(* CODESYS project Almost_done.export

Project tree, tasks and I/O mapping:
  Device : CODESYS Control Win V3 x64, 3S - Smart Software Solutions GmbH, version 3.5.17.0
    application Application
      libraries: Standard, * (System); VisuDialogs, * (System)
      task MainTask (cyclic, interval t#20ms, priority 1) calls PLC_PRG
      task VISU_TASK (cyclic, interval 100 ms, priority 31) calls VisuElems.Visu_Prg
      global variables GVL
      global variables HMI
      global variables OPC
      function block Assembly [ST]
      function block Crane [ST]
      function block ExitMagazine [ST]
      function FillWarehouseArray [ST]
      function FindFreePlace [ST]
      function block PalletizerElevator [ST]
      program PLC_PRG [ST]
      function Round [ST]
      function SetArrayToZero [ST]
      function block ThreeAxis [ST]
      function block TwoAxisLogic [ST]
      function WhereIsMaterial [ST]
      Symbols
      visualisation Assembly
      visualisation Menu
      visualisation Package_Reload
      visualisation Palletizer
      visualisation QA
      visualisation Warehosue_1
      visualisation Warehouse_2
*)

// Device/Application/GVL
VAR_GLOBAL
	Warehouse1Array : ARRAY[1..54] OF BOOL;
	Warehouse1ArrayMaterial  : ARRAY[1..54] OF INT;
	Warehouse2Array : ARRAY[1..54] OF INT ;
	Warehouse2ArrayMaterial  : ARRAY[1..54] OF INT;
	PalletizerArray : ARRAY[0..12] OF BOOL;
END_VAR

// Device/Application/HMI
{attribute 'qualified_only'}
VAR_GLOBAL
	GoingQA : BOOL;
	Emitter1Color : INT := 16;
	Emitter2Color : INT := 16;
	WantedMaterial1 : INT;
	Pick1 : BOOL;
	WantedMaterial2 : INT;
	Pick2 : BOOL;
	ScreenColor : INT := 0;
	EmittMaterials : BOOL := TRUE;
	
	oElevator1Forward : BOOL;
	oPalletizer1Open  : BOOL;
	oPalletizer1Push  : BOOL;
	oPalletizer1Clamp  : BOOL;
	oPalletizer1Forward  : BOOL;
	oPalletizer1ElevatorUp  : BOOL;
	oPalletizer1ChainForward  : BOOL;
	oPalletizer1ElevatorDown : BOOL;
	oPalletizer1ElevatorMoveToMax  : BOOL;
	oPalletizerConv  : BOOL;
	oPalletizerSupplyConv  : BOOL;
	oPalletizerSupplyLightConv  : BOOL;
	oPalletsTowardElevator  : BOOL;
	oPalletizer1Turn  : BOOL;
END_VAR

// Device/Application/OPC
{attribute 'qualified_only'}
VAR_GLOBAL
	// This part includes 2 first machines center and surroundings machines
	iAtAssembledConvEntry : BOOL;
	iAtAssemledPosition : BOOL;
	iMachine1Exit : BOOL;
	iMachine2Exit : BOOL;
	iMachine1Entry : BOOL;
	iMachine2Entry : BOOL;
	iMachiningCenter1Error : BOOL;
	iMachiningCenter2Error : BOOL;
	iMachiningCenter1IsBusy : BOOL;
	iMachiningCenter1Opened : BOOL;
	iMachiningCenter2IsBusy : BOOL;
	iMachiningCenter2Opened : BOOL;
	iMachiningCenter1Progress : DINT;
	iMachiningCenter2Progress : DINT;
	iRightPositioner2Clamped : BOOL;
	iRightPositioner1Clamped : BOOL;
	iRightPositioner1OnPlace : BOOL;
	iRightPositioner2OnPlace : BOOL;
	iRightPositioner3Clamped : BOOL;
	iRightPositioner3OnPlace : BOOL;
	iTwoAxis1Grabbed : BOOL;
	iTwoAxis1MovingX : BOOL;
	iTwoAxis1MovingZ : BOOL;
	iVisionSenserPart1 : DINT;
	iVisionSenserPart2 : DINT;
	
	oAssembledMaterialConv : BOOL;
	oBaseMaterialConv1 : BOOL;
	oBaseMaterialConv2 : BOOL;
	oEmitter1Base : INT;
	oEmitter1Emit : BOOL;
	oEmitter1Part : INT;
	oEmitter2Base : INT;
	oEmitter2Emit : BOOL;
	oEmitter2Part : INT;
	oLiquidMaterialConv1 : BOOL;
	oLiquidMaterialConv2 : BOOL;
	oMachiningCenter1Product : BOOL;
	oMachiningCenter2Product : BOOL;
	oRawMaterialSupply1 : BOOL;
	oRawMaterialSupply2 : BOOL;
	oRightPositioner2Clamp : BOOL;
	oRightPositioner1Clamp : BOOL;
	oRightPositioner1Raise : BOOL;
	oRightPositioner2Raise : BOOL;
	oRightPositioner3Clamp : BOOL;
	oRightPositioner3Raise : BOOL;
	oTwoAxis1X : BOOL;
	oTwoAxis1Z : BOOL;
	oTwoAxis1Grab : BOOL;
	
	//This part include second and third twoAxis pick and place, QA and surroundings conveyors, and first warehouse conveyros
	iAtAssemblyLoadEntry : BOOL;
	iAtCrane1Entry : BOOL;
	iAtCurveConv1Exit : BOOL;
	iAtCurveConv1Entry : BOOL;
	iAtFirstwarehouseCurveConv2Exit : BOOL;
	iAtFirstwarehouseCurveConv2Entry : BOOL;
	iAtPusher : BOOL;
	iAtQACurveEntry : BOOL;
	iAtQAEntry : BOOL;
	iAtQAExit : BOOL;
	iAtWeightConvExit : BOOL;
	iAtWeightConvEntry : BOOL;
	iAtTurntable1Entry : BOOL;
	iAtTurntable1ExitQA : BOOL;
	iAtTurntable1ExitNormal : BOOL;
	iPusher1Back : BOOL;
	iPusher2Back : BOOL;
	iPusher3Back : BOOL;
	iPusher1Front : BOOL;
	iPusher2Front : BOOL;
	iPusher3Front : BOOL;
	iTurntable1Back : BOOL;
	iTurntable1Front : BOOL;
	iTurntable1AtZero : BOOL;
	iTurntable1AtNinety : BOOL;
	iTwoAxis2Grabbed : BOOL;
	iTwoAxis2MovingX : BOOL;
	iTwoAxis3Grabbed : BOOL;
	iTwoAxis3MovingX : BOOL;
	iTwoAxis3MovingZ : BOOL;
	iTwoAxis2MovingZ : BOOL;
	iVisionSensor1 : BOOL;
	iVisionSensor2 : BOOL;
	iWeightConv : REAL;
	iAtQALightConvExit : BOOL;
	iAtElevator2Entry : BOOL;
	iElevator2LeftLimit : BOOL;
	iElevator2RightLimit : BOOL;
	iElevator2CurrentPoint : REAL;
	
	oFirstWarehouseConv1 : BOOL;
	oFirstWarehouseConv3 : BOOL;
	oFirstWarehouseConvLoad : BOOL;
	oFirstWarehouseCurveConv2 : BOOL;
	oPalletAndBoxConv1 : BOOL;
	oPalletAndBoxConv3 : BOOL;
	oPalletAndBoxCurveConv2 : BOOL;
	oPusher1 : BOOL;
	oPusher2 : BOOL;
	oPusher3 : BOOL;
	oQAConv2 : BOOL;
	oQACurveConv : BOOL;
	oQALightConv1 : BOOL;
	oQALightConv2 : BOOL;
	oQALightConv3 : BOOL;
	oQALightConv4 : BOOL;
	oTurntable1Turn : BOOL;
	oTurntable1Forward : BOOL;
	oTurntable1Backward : BOOL;
	oTwoAxis2X : BOOL;
	oTwoAxis2Z : BOOL;
	oTwoAxis3X : BOOL;
	oTwoAxis3Z : BOOL;
	oTwoAxis2Grab : BOOL;
	oTwoAxis3Grab : BOOL;
	oWeightConvBackward : BOOL;
	oWeightConvToward : BOOL;
	oElevator2Forward : BOOL;
	oElevator2SetPoint : REAL;
	oQAConv1 : BOOL;
	
	//This part includes two cranes and conveyor betweeen them
	iAtCrane1Exit : BOOL;
	iAtCrane2Exit : BOOL;
	iAtExitWarehouseExit : BOOL;
	iAtTurntable2Exit : BOOL;
	iAtTurntable2Entry : BOOL;
	iAtTurntable2ExitWarehouse1 : BOOL;
	iAtTurntable2ExitWarehouse2 : BOOL;
	iCrane1AtStart : BOOL;
	iCrane2AtStart : BOOL;
	iCrane1MovingX : BOOL;
	iCrane1MovingZ : BOOL;
	iCrane2MovingX : BOOL;
	iCrane2MovingZ : BOOL;
	iCrane1MidLimit : BOOL;
	iCrane2MidLimit : BOOL;
	iCrane1LeftLimit : BOOL;
	iCrane2LeftLimit : BOOL;
	iCrane1RightLimit : BOOL;
	iCrane2RightLimit : BOOL;
	iTurntable2Back : BOOL;
	iTurntable2Front : BOOL;
	iTurntable2Atzero : BOOL;
	iTurntable2AtNinety : BOOL;
	
	oCrane1Left : BOOL;
	oCrane1Lift : BOOL;
	oCrane2Left : BOOL;
	oCrane2Lift : BOOL;
	oCrane1Right : BOOL;
	oCrane2Right : BOOL;
	oCrane1TargetPosition : INT;
	oCrane2TargetPosition : INT;
	oExitWarehouseConv1 : BOOL;
	oExitWarehouseConv2 : BOOL;
	oFirstWarehouseConvLoadOpposite : BOOL;
	oSecondWarehouseLoadConvOpposite : BOOL;
	oTowardFirstWarehouse : BOOL;
	oTowardSecondWarehouse : BOOL;
	oTurntable2Turn : BOOL;
	oTurntable2Forward : BOOL;
	oTurntable2Backward : BOOL;

	//this part include Box Pick and Place, and conveyors till elevator
	iAtBoxSupplyCurveConv2Exit : BOOL;
	iAtBoxSupplyCurveConv2Entry : BOOL;
	iAtBoxSupplyEnter : BOOL;
	iAtElevatorEntry : BOOL;
	iAtLoadEmptyBoxEntry : BOOL;
	iAtLoadEmptyBoxExit : BOOL;
	iAtPalletDestinationEntry : BOOL;
	iAtPalletDestinationExit : BOOL;
	iAtSecondWarehouseCurveConv3Exit : BOOL;
	iAtSecondWarehouseCurveConv3Entry : BOOL;
	iAtSecondWarehouseConv5 : BOOL;
	iBigBox : BOOL;
	iMidBox : BOOL;
	iPickPlace1Rotated : BOOL;
	iPickPlace1CurrentX : REAL;
	iPickPlace1CurrentY : REAL;
	iPickPlace1CurrentZ : REAL;
	iPickPlace1BoxDetected : BOOL;
	iSmallBox : BOOL;
	
	oBoxSupplyConv1 : BOOL;
	oBoxSupplyConv3 : BOOL;
	oBoxSupplyCurveConv2 : BOOL;
	oEmptyBoxConvSupply : BOOL;
	oPickPlace1X : REAL;
	oPickPlace1Y : REAL;
	oPickPlace1Z : REAL;
	oPickPlace1Grab : BOOL;
	oSecondWarehouseConv1 : BOOL;
	oSecondWarehouseConv12 : BOOL;
	oSecondWarehouseConv2 : BOOL;
	oSecondWarehouseConv4 : BOOL;
	oSecondWarehouseConv5 : BOOL;
	oSecondWarehouseCurveConv3 : BOOL;
	
	//Palletizer
	iAtElevatorUpEntry : BOOL;
	iAtPalletizerChainEntry : BOOL;
	iAtPalletizerConvEntry : BOOL;
	iAtPalletizerEntry : BOOL;
	iPalletizer1Clamped : BOOL;
	iPalletizer1Opening : BOOL;
	iPalletizer1Pushing : BOOL;
	iPalletizer1ElevatorBack : BOOL;
	iPalletizer1ElevatorFront : BOOL;
	iPalletizer1ElevatorMoving : BOOL;
	
	oPalletizer1Open : BOOL;
	oPalletizer1Push : BOOL;
	oPalletizer1Turn : BOOL;
	oPalletizer1Clamp : BOOL;
	oPalletizer1Forward : BOOL;
	oPalletizer1ElevatorUp : BOOL;
	oPalletizer1ChainForward : BOOL;
	oPalletizer1ElevatorDown : BOOL;
	oPalletizer1ChainBackward : BOOL;
	oPalletizer1ElevatorMoveToMax : BOOL;
	oPalletizerConv : BOOL;
	oPalletizerSupplyConv : BOOL;
	oPalletizerSupplyLightConv : BOOL;
	oPalletsTowardElevator : BOOL;
	
	//Elevator near palletizer
	iAtCrane2Entry : BOOL;
	iAtElevatorExit : BOOL;
	iElevator1LeftLimit : BOOL;
	iElevator1RightLimit : BOOL;
	iElevator1CurrentPoint : REAL;
	oElevator1Forward : BOOL;
	oElevator1SetPoint : REAL;
	oSecondWarehouseConv6 : BOOL;
	oSecondWarehouseLoadConv : BOOL;
	
	// Control panel Box Supply
	iBoxSupplyAutomatic : BOOL;
	iBoxSupplyEmergency : BOOL;
	iBoxSupplyManual : BOOL;
	iBoxSupplyStart : BOOL;
	iBoxSupplyStop : BOOL;
	iSafetyDoorBoxSupply : BOOL;
	oBoxSupplyStart : BOOL;
	oBoxSupplyStop : BOOL;
	
	// Control panel palletizer
	iPalletizerAutomatic : BOOL;
	iPalletizerEmergency : BOOL;
	iPalletizerManual : BOOL;
	iPalletizerStart : BOOL;
	iPalletizerStop : BOOL;
	oPalletizerStart : BOOL;
	oPalletizerStop : BOOL;
	
	// Machine center 1 & 2
	oMachiningCenter1Stop : BOOL;
	oMachiningCenter2Stop : BOOL;
	oMachiningCenter1Reset : BOOL;
	oMachiningCenter1Start : BOOL;
	oMachiningCenter2Reset : BOOL;
	oMachiningCenter2Start : BOOL;
	
	// Control panel Assembly
	iAssemblyAutomatic : BOOL;
	iAssemblyEmergency : BOOL;
	iAssemblyManual : BOOL;
	iAssemblyStart : BOOL;
	iAssemblyStop : BOOL;
	oAssemblyStart : BOOL;
	oAssemblyStop : BOOL;
	
END_VAR

// Device/Application/PLC_PRG
PROGRAM PLC_PRG
VAR
	ONE : INT := 1;
	TWO : INT := 2;
	TwoAxis13Array : ARRAY[0..8] OF INT := [1,3,2,1,3,4,0,0];
	TwoAxis2Array  : ARRAY[0..8] OF INT := [2,1,3,4,1,3,0,1];
	QAArray : ARRAY[0..99, 0..2] OF INT;
	ExitMagazine12 : ExitMagazine;
	Crane1DesignedLocation : INT;
	PackageOnPlace : BOOL;
	Crane1 : Crane;
	Crane2 : Crane;
	ThreeAxis1 : ThreeAxis;
	PalletizerElevator1 : PalletizerElevator;
	Crane1Working : BOOL;
	Crane1Swap : BOOL;
	QABoxNumber : INT;
	QABusy : BOOL;
	QAMaterialNumber : INT;
	MaterialnBox : CTU;
	Timer1Logic : BOOL;
	Timer1 : TON;
	MaterialsPicked : CTU;
	RaisePositioner2 : BOOL;
	QALightConv1 : BOOL;
	QALightConv234 : BOOL;
	F_QALightConvExit : F_TRIG;
	FirstWarehouseConv1 : BOOL;
	Push1 : BOOL;
	Push2 : BOOL;
	Push3 : BOOL;
	Counter1 : CTUD;
	Counter2 : CTUD;
	F_WeightConvEntry : F_TRIG;
	F_WeightConvExit : F_TRIG;
	R_Pusher1 : R_TRIG;
	R_Pusher2 : R_TRIG;
	R_Pusher3 : R_TRIG;
	CurveArray1 : CTUD;
	CurveConv2 :  CTUD;
	NotCurveConvExit : BOOL;
	NotCurveExit : BOOL;
	PackageReady : BOOL;
	R_CurveConv2Exit : R_TRIG;
	F_Cran1Entry : F_TRIG;
	FirstWarehouseConv3 : BOOL;
	TwoAxis1 : TwoAxisLogic;
	TwoAxis2 : TwoAxisLogic;
	TwoAxis3 : TwoAxisLogic;
	LiquidMaterialConv1: BOOL;
	BaseMaterialConv1 : BOOL;
	R_MachineCenter1Working : R_TRIG;
	F_PalletEntryTwoAxis2   : F_TRIG;
	R_QAConv   : R_TRIG;
	F_QAEntry : F_TRIG;
	QAConvWorking : BOOL;
	VisionSensor1        : BOOL := FALSE;
	VisionSensor2        : BOOL := FALSE;
	AssemblyMaterialMove : BOOL;
	F_VisionSensor1 	 : F_TRIG;
	F_VisionSensor2 	 : F_TRIG;
	F_AssemblyExit 	 	 : F_TRIG;
	F_Turntable1ExitQA 	 : F_TRIG;
	F_Turntable1ExitNormal : F_TRIG;
	R_Turntable1Front    : R_TRIG;
	Turn1Logic 			 : BOOL;
	TwoAxis1Working 	 : BOOL;
	TwoAxis2Working		 : BOOL;
	TwoAxis3Working 	 : BOOL;
	TwoAxis2WorkingPosition : BOOL;
	TwoAxis2MaterialReady : BOOL;
	TwoAxis3WorkingPosition : BOOL;
	Part1Ready : BOOL;
	Part2Ready : BOOL;
	Clamping1 : BOOL;
	Clamping2 : BOOL;
	Clamping3 : BOOL;
	TwoAxis1MoveDown : BOOL;
	TwoAxis1MoveUp : BOOL;
	TwoAxis1MoveForward : BOOL;
	TwoAxis1MoveBackward : BOOL;
	TwoAxis1Grabbed : BOOL;
	TwoAxis1Done : BOOL;
	AssemblyConvMove : BOOL;
	F_AssembledPosition : F_TRIG;
	PalletAndBoxConv3 : BOOL;
	Turntable1Forward : BOOL;
	R_ExitElevator : R_TRIG;
	F_Warehouse2Entry : F_TRIG;
	PalletOnPlace : BOOL := FALSE;
	PalletReady : BOOL;
	Crane2DesignedLocation : INT;
	Crane2Working : BOOL;
	Crane2Swap : BOOL;
	LastPart : CTUD;
	ElevatorBusy : BOOL;
	NotExit : BOOL;
	StartTwoAxis3 : TON;
	TimeHolder : BOOL;
	RealHighElevator2 : REAL;
	R_Elevator2Entry : R_TRIG;
	F_InElevator2 : F_TRIG;
	QAWaiting : BOOL;
	Forward2 : BOOL;
	QAConvWorking2 : BOOL;
END_VAR

(* Logic behind Machine Center 1 *)

// Emitter should always be true, changing it's color will be done from HMIs
OPC.oEmitter1Emit := TRUE;
OPC.oEmitter1Part := HMI.Emitter1Color;
// Conv supply should send raw material only when machine 1 center not busy and there is no raw material at entry
OPC.oRawMaterialSupply1 := NOT OPC.iMachine1Entry AND NOT OPC.iMachiningCenter1IsBusy;
// Machine Center should start working as soon as there is raw material in
OPC.oMachiningCenter1Start := OPC.iMachine1Entry;

(* Logic behind Machine Center 2 *)

// Emitter should always be true, changing it's color will be done from HMI
OPC.oEmitter2Emit := TRUE;
OPC.oEmitter2Part := HMI.Emitter2Color;
// We want to make second part of material so we must change this variable to true
OPC.oMachiningCenter1Product := TRUE;
OPC.oMachiningCenter2Product := FALSE;
// Conv supply should send raw material only when machine 2 center not busy and there is no raw material at entry
OPC.oRawMaterialSupply2 := NOT OPC.iMachine2Entry AND NOT OPC.iMachiningCenter2IsBusy;
// Machine Center should start working as soon as there is raw material in
OPC.oMachiningCenter2Start := OPC.iMachine2Entry;

(* Converoys from Machine center *)

// At first we want to make CTUD counter which will count how many parts are in move
Counter1(CU := OPC.iMachine1Exit, CD:= VisionSensor1);
Counter2(CU := OPC.iMachine2Exit, CD:= VisionSensor2);

// Now when we have our counter, if the CV is bigger than 0, QD whille be false so we have mocing part
LiquidMaterialConv1 := NOT Counter2.QD;

// Same as above, if CV bigger than 0, conv should move if possible
BaseMaterialConv1 := NOT Counter1.QD;

// When should move conveyors from machine center 2
OPC.oLiquidMaterialConv1 := OPC.oLiquidMaterialConv2 AND LiquidMaterialConv1 ;
OPC.oLiquidMaterialConv2 := NOT TwoAxis1Working OR AssemblyMaterialMove;

// When should move conveyors from machine center 1
OPC.oBaseMaterialConv1 := OPC.oBaseMaterialConv2 AND BaseMaterialConv1 ;
OPC.oBaseMaterialConv2 := NOT TwoAxis1Working;

(* Two Axis Pick & Place which assemble two parts, two vision sensors, two right positioners and  light conv behind them *)

// At first we want to make falling trigger using vision senser, those numbers are taken from factory i/o
IF OPC.iVisionSenserPart1 = 2 OR OPC.iVisionSenserPart1 = 5 OR OPC.iVisionSenserPart1 = 8 THEN
	VisionSensor1 := TRUE;
ELSE 
	VisionSensor1 := FALSE;
END_IF;

// Same as previous we want to check when expected material went in
IF OPC.iVisionSenserPart2 = 3 OR OPC.iVisionSenserPart2 = 6 OR OPC.iVisionSenserPart2 = 9 THEN
	VisionSensor2 := TRUE;
ELSE 
	VisionSensor2 := FALSE;
END_IF;

// Making falling trigger 
F_VisionSensor1(CLK := VisionSensor1);
F_VisionSensor2(CLK := VisionSensor2);

// Checking if the parts are on positon, then clamping them
IF F_VisionSensor1.Q THEN 
	Clamping1 := TRUE;
	OPC.oRightPositioner1Clamp := TRUE;
END_IF;

// Checking if clamped
IF Clamping1 AND OPC.iRightPositioner1Clamped THEN
	Part1Ready := TRUE;
	OPC.oRightPositioner1Clamp := FALSE;
	Clamping1 := FALSE;
END_IF;

// Now the very same thing for second positioner

// Checking if the parts are on positon, then clamping them
IF F_VisionSensor2.Q THEN 
	Clamping2 := TRUE;
	OPC.oRightPositioner2Clamp := TRUE;
END_IF;

// Checking if clamped
IF Clamping2 AND OPC.iRightPositioner2Clamped THEN
	Part2Ready := TRUE;
	//OPC.oRightPositioner2Clamp := FALSE;
	Clamping2 := FALSE;
END_IF;

// If both parts are ready, two axis pick and place will assembly them, at first it will move down to take first part
IF Part1Ready AND Part2Ready THEN
	TwoAxis1Working := TRUE;
	Part2Ready := FALSE;
	Part1Ready := FALSE;
END_IF;

// Using FB to pick and plice material
TwoAxis1( Start:= TwoAxis1Working, IncomingArray := TwoAxis13Array, Grabbed := OPC.iTwoAxis1Grabbed, MovingX := OPC.iTwoAxis1MovingX, MovingZ := OPC.iTwoAxis1MovingZ);
OPC.oTwoAxis1X := TwoAxis1.X;
OPC.oTwoAxis1Z := TwoAxis1.Z;
OPC.oTwoAxis1Grab := TwoAxis1.Grab;

// Set working variable to 0 and raise the positioner
IF TwoAxis1.JobDone THEN
	TwoAxis1Working := FALSE;
	RaisePositioner2 := TRUE;
	OPC.oRightPositioner2Clamp := FALSE; // It wasnt here befor, just to check if this will work
END_IF;

// IF assemby done, then open right positioner 2
OPC.oRightPositioner2Raise := RaisePositioner2;

// When right positioner is up, move material
IF RaisePositioner2 AND  OPC.iRightPositioner1OnPlace THEN
	AssemblyMaterialMove := TRUE;
END_IF;

// Close opened right positioner 2
F_AssemblyExit(CLK := OPC.iAtAssembledConvEntry);
IF F_AssemblyExit.Q THEN
	OPC.oRightPositioner1Raise := FALSE;
	AssemblyMaterialMove := FALSE;
	AssemblyConvMove := TRUE;
	RaisePositioner2 := FALSE;
END_IF;

// Falling trigger at the end of this conv
F_AssembledPosition(CLK := OPC.iAtAssemledPosition);

// When f_trig at the end, stop conveyor
IF F_AssembledPosition.Q THEN
	AssemblyConvMove := FALSE;
	Clamping3 := TRUE;
	OPC.oRightPositioner3Clamp := TRUE;
END_IF;

// Clamp material to desired position
IF Clamping3 AND OPC.iRightPositioner3Clamped THEN
	Clamping3 := FALSE;
	TwoAxis2MaterialReady := TRUE;
	OPC.oRightPositioner3Clamp := FALSE;
END_IF;

// Logic when should this conv move
OPC.oAssembledMaterialConv := AssemblyConvMove OR OPC.iAtAssembledConvEntry;

(* Logic when should second pick and place take the assembled material *)

//Making rising triggerws which will inform us weather there is pallet in determined place
F_PalletEntryTwoAxis2(CLK := OPC.iAtAssemblyLoadEntry);
// When pallet is on place we set two axis pick place in working stance, now we wait for materials
IF F_PalletEntryTwoAxis2.Q THEN
	TwoAxis2WorkingPosition := TRUE;
END_IF;
// At first we have to move coveroy which send the pallet wuth the box, we usually want it to run when there is no pallet on determined place
OPC.oPalletAndBoxConv1 := NOT TwoAxis2WorkingPosition;

// When should two axis 2 work 
IF TwoAxis2WorkingPosition AND TwoAxis2MaterialReady THEN
	TwoAxis2Working := TRUE;
	TwoAxis2MaterialReady := FALSE;
END_IF;

// Calling FB which will take the element and place it in the box
TwoAxis2( Start:= TwoAxis2Working, IncomingArray := TwoAxis2Array, Grabbed := OPC.iTwoAxis2Grabbed, MovingX := OPC.iTwoAxis2MovingX, MovingZ := OPC.iTwoAxis2MovingZ);
OPC.oTwoAxis2X := TwoAxis2.X;
OPC.oTwoAxis2Z := TwoAxis2.Z;
OPC.oTwoAxis2Grab := TwoAxis2.Grab;


// When job is done we set variable back to 0
IF TwoAxis2.JobDone THEN
	TwoAxis2Working := FALSE;
END_IF;

// Now we would like to count how many things we have in box
MaterialnBox(CU := TwoAxis2.JobDone, PV := 3);

// If we've got 3 materials in box we set the box out
IF MaterialnBox.Q THEN
	TwoAxis2WorkingPosition := FALSE;
END_IF;
MaterialnBox.RESET := MaterialnBox.Q;

(* This part is about sending box either to QA or Magazine *)

// We would like to use counter in order to power conveyor, but cu and cd require raising trigger so we need to invert one variable
NotCurveExit := NOT OPC.iAtCurveConv1Exit;

// Counter
CurveArray1(CU := OPC.iAtCurveConv1Entry, CD:= NotCurveExit);

// If there is more than one pallet, simply power the curve conveyor
OPC.oPalletAndBoxCurveConv2 := NOT CurveArray1.QD;


// Long conv before first turntable
IF OPC.iAtCurveConv1Exit THEN
	PalletAndBoxConv3 := TRUE;
END_IF

// When should move conveoyr before turn table 1
OPC.oPalletAndBoxConv3 := PalletAndBoxConv3 AND(NOT OPC.iAtTurntable1Entry OR OPC.iTurntable1AtZero);

// Move pallet to the middle of turn table
IF OPC.iAtTurntable1Entry THEN
	Turntable1Forward := TRUE;
END_IF;

// Rising trigger, If at middle, set to false both conveyros and turn
R_Turntable1Front(CLK := OPC.iTurntable1Front); 

// When package is on the front we want to stop conveyors and rotate it
IF R_Turntable1Front.Q THEN
	Turntable1Forward := FALSE;
	PalletAndBoxConv3 := FALSE;
	Turn1Logic := TRUE;
END_IF

// Tabl;e should turn when rising trigger fornt sensor
OPC.oTurntable1Turn := Turn1Logic;

// Making 2 falling triggers which inform us when pallet lefts table
F_Turntable1ExitQA(CLK := OPC.iAssemblyAutomatic);
F_Turntable1ExitNormal(CLK := OPC.iAtTurntable1ExitNormal);

// IF left turn table, return to normal
IF F_Turntable1ExitQA.Q OR F_Turntable1ExitNormal.Q THEN
	Turn1Logic := FALSE;
END_IF;

// If turned and going to QA, goo left
OPC.oTurntable1Forward := (HMI.GoingQA AND OPC.iTurntable1AtNinety) OR Turntable1Forward;

// If turned and going warehouse, charge right
OPC.oTurntable1Backward := NOT HMI.GoingQA AND OPC.iTurntable1AtNinety;

// Raising trigger to power our conveyor
R_QAConv(CLK := OPC.iAtTurntable1ExitQA);

// IF raising trigger then change variable which move conv
IF R_QAConv.Q THEN
	QAConvWorking := TRUE;
END_IF;

// Conveor moves when QAConvWorking from raising trigger true
OPC.oQAConv1 := QAConvWorking AND (NOT OPC.iAtElevator2Entry OR RealHighElevator2 = 0.0);

RealHighElevator2 := Round(First := OPC.iElevator2CurrentPoint);

// Falling trigger to stop our conv
F_QAEntry(CLK := OPC.iAtQAEntry);

R_Elevator2Entry(CLK := OPC.iAtElevator2Entry);
F_InElevator2(CLK := OPC.iElevator2RightLimit);

IF R_Elevator2Entry.Q THEN
	QAWaiting := TRUE;
END_IF

IF QAWaiting AND RealHighElevator2 = 0.0 THEN
	Forward2 := TRUE;
END_IF

IF F_InElevator2.Q THEN
	Forward2 := FALSE;
	OPC.oElevator2SetPoint := 0.35; 
END_IF

IF RealHighElevator2 = 0.35 THEN
	Forward2 := TRUE;
	QAConvWorking2 := TRUE;
END_IF

OPC.oQAConv2 := QAConvWorking2;
OPC.oElevator2Forward := Forward2;

// When pallet on it;s place, stop it
IF F_QAEntry.Q THEN
	HMI.GoingQA := FALSE;
	QAConvWorking2 := FALSE;
	TwoAxis3WorkingPosition := TRUE;
	OPC.oElevator2SetPoint := 0.0;
END_IF;

// Instance of FB which operate our two axis
TwoAxis3( Start:= TwoAxis3Working, IncomingArray := TwoAxis13Array, Grabbed := OPC.iTwoAxis3Grabbed, MovingX := OPC.iTwoAxis3MovingX, MovingZ := OPC.iTwoAxis3MovingZ);
OPC.oTwoAxis3X := TwoAxis3.X;
OPC.oTwoAxis3Z := TwoAxis3.Z;
OPC.oTwoAxis3Grab := TwoAxis3.Grab;

// Setting counter which will tell us how many material have been picked
MaterialsPicked( CU := TwoAxis3.JobDone, PV := 3);
IF MaterialsPicked.CV >= 100 THEN
	ONE := 100; /////jest check
END_IF

// If 3 or more materials picked stop working at this moment, pallet will be pushed next with next pallet entry
IF MaterialsPicked.Q THEN
	TwoAxis3WorkingPosition := FALSE;
END_IF;
MaterialsPicked.RESET := MaterialsPicked.Q;

// When job done set to false, in order to reset pick up cycle
IF TwoAxis3.JobDone THEN
	TimeHolder := FALSE;
	QALightConv1 := TRUE;
END_IF;
 
// when robot should be working and he's not working(which means he finished one run) run it again
IF TwoAxis3WorkingPosition AND NOT TwoAxis3Working THEN
	TimeHolder := TRUE;
END_IF

StartTwoAxis3(IN := TimeHolder, PT := T#2000MS);
TwoAxis3Working := StartTwoAxis3.Q;

// Logic when should move first QA conv
OPC.oQALightConv1 := QALightConv1 AND (NOT OPC.iAtWeightConvEntry OR NOT QABusy);

// Making falling trigger which tells us when our material enter weight conv
F_WeightConvEntry(CLK := OPC.iAtWeightConvEntry);

// When our material fully enter weight conv we would like to stop it
IF F_WeightConvEntry.Q THEN
	Timer1Logic := TRUE;
	QALightConv1 := FALSE;
	QABusy := TRUE;
END_IF;

// Logic when should weight conv charge forward
OPC.oWeightConvToward := Timer1.Q OR OPC.iAtWeightConvEntry;

// here we would like to save our readings, not sure how right now
IF Timer1.ET > T#1S THEN
	// !!!!!!!!!!!! THIS IS JUST A FILLER, LATER WHEN WE FIGURE OUT HOW TO DO IT WE WILL DO IT
	QAArray[QABoxNumber, QAMaterialNumber] := 4 ;
END_IF;

// timer 1, we need to read analog reading when conv doesnt move so we stop conv and after 2s we want to varge forward
Timer1(IN:= Timer1Logic, PT := T#2S);

// falling trigger which tell us when material leaves weight conv
F_WeightConvExit(CLK := OPC.iAtWeightConvExit);

// When material left weight conv simply stop charging forward
IF F_WeightConvExit.Q THEN
	Timer1Logic := FALSE;
	QALightConv234 := TRUE;
END_IF;

// Checnking when wrong matterial entered the yeet position
R_Pusher1(CLK := OPC.iAtPusher);
R_Pusher2(CLK := OPC.iVisionSensor1); 
R_Pusher3(CLK := OPC.iVisionSensor2); 

// Logic when should pusheers work,
IF R_Pusher1.Q AND QAArray[QABoxNumber, QAMaterialNumber] = 4 THEN
	Push1 := TRUE;
	QALightConv234 := FALSE;
ELSIF OPC.iPusher1Front THEN
	Push1 := FALSE;
END_IF
// same as above
IF R_Pusher2.Q THEN
	Push2 := TRUE;
	QALightConv234 := FALSE;
ELSIF OPC.iPusher2Front THEN
	Push2 := FALSE;
END_IF
// same as above
IF R_Pusher3.Q THEN
	Push3 := TRUE;
	QALightConv234 := FALSE;
ELSIF OPC.iPusher3Front THEN
	Push3 := FALSE;
END_IF

// Falling trigger which tells us when material leaves conv
F_QALightConvExit(CLK := OPC.iAtQALightConvExit);

// when material leaves conv we would like to stop convs
IF F_QALightConvExit.Q THEN
	QALightConv234 := FALSE;
END_IF;

// Assigment pushers logic to variables declared earlier
OPC.oPusher3 := Push3;
OPC.oPusher2 := Push2;
OPC.oPusher1 := Push1;

// Multiple assigment to control all light conveyors in QA
OPC.oQALightConv4 := OPC.oQALightConv3 := OPC.oQALightConv2 := QALightConv234;

// Launch conveyor when material is on the way
IF F_Turntable1ExitNormal.Q THEN
	FirstWarehouseConv1 := TRUE;
END_IF

// Logic when should conv move, move when box on sensor or material left sensor and there is no package awaiting
OPC.oFirstWarehouseConv1 := (FirstWarehouseConv1 OR OPC.iAtTurntable1ExitNormal) AND (NOT PackageOnPlace OR NOT OPC.iAtFirstwarehouseCurveConv2Entry) ;

// making inverse vairable so we can make F_trig into R_trig in ctud below
NotCurveConvExit := NOT OPC.iAtFirstwarehouseCurveConv2Exit;
// Counter which counter how many matterials have entered and left this conv
CurveConv2(CU:= OPC.iAtFirstwarehouseCurveConv2Entry, CD:= NotCurveConvExit);

// When 0 on CTUD above, that means there is no material on this conv, as well we dont want it to move if package await
OPC.oFirstWarehouseCurveConv2 := NOT CurveConv2.QD AND(NOT PackageOnPlace OR NOT OPC.iAtFirstwarehouseCurveConv2Exit);

// When material arrives on last conv before warehguse
R_CurveConv2Exit(CLK := OPC.iAtFirstwarehouseCurveConv2Exit);

// IF there is material on front we change variable which move conv
IF R_CurveConv2Exit.Q THEN
	FirstWarehouseConv3 := TRUE;
END_IF

// When material reach designed place we want it to stop conv and prepare crane 
F_Cran1Entry(CLK := OPC.iAtCrane1Entry);
// as above, when material arrive we want to stop conv and launch crane 1
IF F_Cran1Entry.Q THEN
	FirstWarehouseConv3 := FALSE;
	PackageOnPlace:= TRUE;
END_IF;

IF NOT Crane1.Working AND PackageOnPlace THEN
	PackageOnPlace:= FALSE;
	PackageReady := TRUE;
END_IF;

// Logic behind controlling conv before warehouse

//OPC.oFirstWarehouseConv3 := FirstWarehouseConv3 AND NOT PackageReady;
OPC.oFirstWarehouseConv3 := FirstWarehouseConv3;
OPC.oFirstWarehouseConvLoad := FirstWarehouseConv3;

IF PackageReady THEN
	Crane1DesignedLocation := FindFreePlace(ONE);
	IF Crane1DesignedLocation  <> 0 THEN
		PackageReady := FALSE;
		Crane1Working := TRUE;
	ELSE 
		PackageReady := FALSE;
		Crane1Swap := TRUE;
	END_IF
END_IF
Crane1(LeftOrRight := FALSE, Swap := Crane1Swap, Place := Crane1Working, Pick := HMI.Pick1, CraneLeftLimit := OPC.iCrane1LeftLimit,
CraneRightLimit := OPC.iCrane1RightLimit, CraneMidLimit := OPC.iCrane1MidLimit, CraneMovingZ := OPC.iCrane1MovingZ,
CraneMovingX := OPC.iCrane1MovingX, CraneAtStart := OPC.iCrane1AtStart,
WantedMaterial := HMI.WantedMaterial1, WarehouseNumer := 1, CanEnd := OPC.iAtCrane1Exit);

	OPC.oCrane1TargetPosition := Crane1.CraneTargetPosition; 
	OPC.oCrane1Right := Crane1.CraneRight ;
	OPC.oCrane1Left := Crane1.CraneLeft ;
	OPC.oCrane1Lift := Crane1.CraneLift ;
	IF Crane1.Working THEN 
		Crane1Working := FALSE;
		Crane1Swap := FALSE;
	END_IF


ExitMagazine12(iAtCrane1Exit := OPC.iAtCrane1Exit, iAtCrane2Exit := OPC.iAtCrane2Exit, iAtExitWarehouseExit := OPC.iAtExitWarehouseExit,
iAtTurntable2Exit := OPC.iAtTurntable2Exit, iAtTurntable2Entry := OPC.iAtTurntable2Entry,
iAtTurntable2ExitWarehouse1 := OPC.iAtTurntable2ExitWarehouse1, iAtTurntable2ExitWarehouse2 := OPC.iAtTurntable2ExitWarehouse2,
iTurntable2Back := OPC.iTurntable2Back, iTurntable2Front := OPC.iTurntable2Front, iTurntable2Atzero := OPC.iTurntable2Atzero,
iTurntable2AtNinety := OPC.iTurntable2AtNinety);

	OPC.oExitWarehouseConv1 := ExitMagazine12.oExitWarehouseConv1;
	OPC.oExitWarehouseConv2 := ExitMagazine12.oExitWarehouseConv2;
	OPC.oFirstWarehouseConvLoadOpposite := ExitMagazine12.oFirstWarehouseConvLoadOpposite;
	OPC.oSecondWarehouseLoadConvOpposite := ExitMagazine12.oSecondWarehouseLoadConvOpposite;
	OPC.oTowardSecondWarehouse := ExitMagazine12.oTowardSecondWarehouse;
	OPC.oTurntable2Forward :=  ExitMagazine12.oTurntable2Forward;
	OPC.oTurntable2Backward := ExitMagazine12.oTurntable2Backward;
	OPC.oTurntable2Turn := ExitMagazine12.oTurntable2Turn;


ThreeAxis1(iBoxSupplyStart := OPC.iBoxSupplyStart, iBoxSupplyStop := OPC.iBoxSupplyStop, iSafetyDoorBoxSupply := OPC.iSafetyDoorBoxSupply,
iBigBox := OPC.iBigBox, iMidBox := OPC.iMidBox, iSmallBox := OPC.iSmallBox, iAtBoxSupplyEnter := OPC.iAtBoxSupplyEnter,
iAtBoxSupplyCurveConv2Entry := OPC.iAtBoxSupplyCurveConv2Entry, iAtBoxSupplyCurveConv2Exit := OPC.iAtBoxSupplyCurveConv2Exit,
iAtPalletDestinationEntry := OPC.iAtPalletDestinationEntry, iAtPalletDestinationExit := OPC.iAtPalletDestinationExit,
iAtLoadEmptyBoxEntry := OPC.iAtLoadEmptyBoxEntry, iAtLoadEmptyBoxExit := OPC.iAtLoadEmptyBoxExit,
iAtSecondWarehouseCurveConv3Entry := OPC.iAtSecondWarehouseCurveConv3Entry, iPickPlace1Rotated := OPC.iPickPlace1Rotated,
iPickPlace1CurrentX := OPC.iPickPlace1CurrentX, iPickPlace1CurrentY := OPC.iPickPlace1CurrentY,
iPickPlace1CurrentZ := OPC.iPickPlace1CurrentZ, iPickPlace1BoxDetected := OPC.iPickPlace1BoxDetected,
iAtSecondWarehouseCurveConv3Exit := OPC.iAtSecondWarehouseCurveConv3Exit, iAtElevatorEntry := OPC.iAtElevatorEntry,
iElevator1CurrentPoint := OPC.iElevator1CurrentPoint, iAtSecondWarehouseConv5 := OPC.iAtSecondWarehouseConv5,
ElevatorBusy := ElevatorBusy);

	OPC.oBoxSupplyConv1 := ThreeAxis1.oBoxSupplyConv1;
	OPC.oBoxSupplyConv3 := ThreeAxis1.oBoxSupplyConv3;
	OPC.oBoxSupplyCurveConv2 := ThreeAxis1.oBoxSupplyCurveConv2;
	OPC.oEmptyBoxConvSupply := ThreeAxis1.oEmptyBoxConvSupply;
	OPC.oPickPlace1X  := ThreeAxis1.oPickPlace1X;
	OPC.oPickPlace1Y  := ThreeAxis1.oPickPlace1Y;
	OPC.oPickPlace1Z  := ThreeAxis1.oPickPlace1Z;
	OPC.oPickPlace1Grab  := ThreeAxis1.oPickPlace1Grab;
	OPC.oSecondWarehouseConv1  := ThreeAxis1.oSecondWarehouseConv1;
	OPC.oSecondWarehouseConv2  := ThreeAxis1.oSecondWarehouseConv2;
	OPC.oSecondWarehouseCurveConv3  := ThreeAxis1.oSecondWarehouseCurveConv3;
	OPC.oSecondWarehouseConv4  := ThreeAxis1.oSecondWarehouseConv4;
	OPC.oSecondWarehouseConv5  := ThreeAxis1.oSecondWarehouseConv5;
	OPC.oSecondWarehouseConv12 := ThreeAxis1.oSecondWarehouseConv12;

PalletizerElevator1(iPalletizerStart := OPC.iPalletizerStart, iPalletizerStop := OPC.iPalletizerStop,
iAtElevatorUpEntry := OPC.iAtElevatorUpEntry, iAtElevatorExit := OPC.iAtElevatorExit, iAtElevatorEntry := OPC.iAtElevatorEntry,
iElevator1RightLimit := OPC.iElevator1RightLimit, iElevator1LeftLimit := OPC.iElevator1LeftLimit,
iElevator1CurrentPoint := OPC.iElevator1CurrentPoint, iPalletizer1ElevatorMoving := OPC.iPalletizer1ElevatorMoving,
iAtPalletizerConvEntry := OPC.iAtPalletizerConvEntry, iAtPalletizerChainEntry := OPC.iAtPalletizerChainEntry,
iPalletizer1ElevatorBack := OPC.iPalletizer1ElevatorBack, iPalletizer1ElevatorFront := OPC.iPalletizer1ElevatorFront,
iAtPalletizerEntry := OPC.iAtPalletizerEntry, iPalletizer1Clamped := OPC.iPalletizer1Clamped, 
iPalletizer1Pushing := OPC.iPalletizer1Pushing,iPalletizer1Opening := OPC.iPalletizer1Opening,
iPalletizerEmergency := OPC.iPalletizerEmergency,iPalletizerAutomatic := OPC.iPalletizerAutomatic,
iPalletizerManual := OPC.iPalletizerManual);
 
	OPC.oElevator1Forward := PalletizerElevator1.oElevator1Forward ;
	OPC.oElevator1SetPoint  := PalletizerElevator1.oElevator1SetPoint;
	OPC.oPalletizer1Open  := PalletizerElevator1.oPalletizer1Open;
	OPC.oPalletizer1Push  := PalletizerElevator1.oPalletizer1Push;
	OPC.oPalletizer1Clamp  := PalletizerElevator1.oPalletizer1Clamp;
	OPC.oPalletizer1Forward  := PalletizerElevator1.oPalletizer1Forward;
	OPC.oPalletizer1ElevatorUp := PalletizerElevator1.oPalletizer1ElevatorUp;
	OPC.oPalletizer1ChainForward := PalletizerElevator1.oPalletizer1ChainForward;
	OPC.oPalletizer1ElevatorDown  := PalletizerElevator1.oPalletizer1ElevatorDown;
	OPC.oPalletizer1ChainBackward  := PalletizerElevator1.oPalletizer1ChainBackward;
	OPC.oPalletizer1ElevatorMoveToMax  := PalletizerElevator1.oPalletizer1ElevatorMoveToMax;
	OPC.oPalletizerConv  := PalletizerElevator1.oPalletizerConv;
	OPC.oPalletizerSupplyConv  := PalletizerElevator1.oPalletizerSupplyConv;
	OPC.oPalletizerSupplyLightConv  := PalletizerElevator1.oPalletizerSupplyLightConv;
	OPC.oPalletsTowardElevator  := PalletizerElevator1.oPalletsTowardElevator;
	OPC.oPalletizer1Turn := PalletizerElevator1.oPalletizer1Turn;
	ElevatorBusy := PalletizerElevator1.ElevatorBusy;
 
 NotExit := NOT OPC.iAtCrane2Entry;
 LastPart(CU := OPC.iAtElevatorExit, CD := NotExit);
 OPC.oSecondWarehouseLoadConv := OPC.oSecondWarehouseConv6 := NOT LastPart.QD AND NOT PalletOnPlace;
 
 F_Warehouse2Entry(CLK := OPC.iAtCrane2Entry);
 IF F_Warehouse2Entry.Q THEN
	 PalletOnPlace := TRUE;
 END_IF
 
 IF PalletOnPlace AND NOT Crane2.Working THEN
	 PalletReady := TRUE;
	 PalletOnPlace := FALSE;
 END_IF
 
 IF PalletReady THEN
	 Crane2DesignedLocation := FindFreePlace(TWO);
	IF Crane2DesignedLocation  <> 0 THEN
		PalletReady := FALSE;
		Crane2Working := TRUE;
	ELSE 
		PalletReady := FALSE;
		Crane2Swap := TRUE;
	END_IF
 END_IF

Crane2(LeftOrRight := TRUE, Swap := Crane2Swap, Place := Crane2Working, Pick := HMI.Pick2, CraneLeftLimit := OPC.iCrane2LeftLimit,
CraneRightLimit := OPC.iCrane2RightLimit, CraneMidLimit := OPC.iCrane2MidLimit, CraneMovingZ := OPC.iCrane2MovingZ,
CraneMovingX := OPC.iCrane2MovingX, CraneAtStart := OPC.iCrane2AtStart,
WantedMaterial := HMI.WantedMaterial2, WarehouseNumer := 2, CanEnd := OPC.iAtCrane2Exit);

	OPC.oCrane2TargetPosition := Crane2.CraneTargetPosition; 
	OPC.oCrane2Right := Crane2.CraneRight ;
	OPC.oCrane2Left := Crane2.CraneLeft ;
	OPC.oCrane2Lift := Crane2.CraneLift ;
	IF Crane2.Working THEN 
		Crane2Working := FALSE;
		Crane2Swap := FALSE;
	END_IF

END_PROGRAM

// Device/Application/Assembly
FUNCTION_BLOCK Assembly
VAR_INPUT
	iMachine1Entry : BOOL;
	iMachine1Exit : BOOL;
	iAtAssembledConvEntry : BOOL;
	iMachine2Exit : BOOL;
	iMachine2Entry : BOOL;
	iAtAssemledPosition : BOOL;
	iRightPositioner1Clamped : BOOL;
	iRightPositioner1OnPlace : BOOL;
	iRightPositioner2Clamped : BOOL;
	iRightPositioner2OnPlace : BOOL;
	iMachiningCenter2IsBusy : BOOL;
	iMachiningCenter1IsBusy : BOOL;
	iVisionSenserPart1 : INT;
	iVisionSenserPart2 : INT;
END_VAR
VAR_OUTPUT
	oAssembledMaterialConv : BOOL;
	oBaseMaterialConv1 : BOOL;
	oBaseMaterialConv2 : BOOL;
	oEmitter1Emit : BOOL;
	oEmitter1Part : INT;
	oEmitter2Emit : BOOL;
	oEmitter2Part : INT;
	oLiquidMaterialConv1 : BOOL;
	oLiquidMaterialConv2 : BOOL;
	oMachiningCenter1Stop : BOOL;
	oMachiningCenter2Stop : BOOL;
	oMachiningCenter1Reset : BOOL;
	oMachiningCenter1Start : BOOL;
	oMachiningCenter2Reset : BOOL;
	oMachiningCenter2Start : BOOL;
	oRawMaterialSupply1 : BOOL;
	oRawMaterialSupply2 : BOOL;
	oRightPositioner1Clamp : BOOL;
	oRightPositioner1Raise : BOOL;
	oRightPositioner2Clamp : BOOL;
	oRightPositioner2Raise : BOOL;
	oMachiningCenter2Product : BOOL;
	oMachiningCenter1Product : BOOL;
	oRightPositioner3Clamp : BOOL;
END_VAR
VAR
	Start : BOOL;
	TwoAxis1 : TwoAxisLogic;
	RaisePositioner2 : BOOL;
	Part1Ready : BOOL;
	Part2Ready : BOOL;
	Counter1 : CTUD;
	Counter2 : CTUD;
	LiquidMaterialConv1: BOOL;
	BaseMaterialConv1 : BOOL;
	R_MachineCenter1Working : R_TRIG;
	VisionSensor1        : BOOL := FALSE;
	VisionSensor2        : BOOL := FALSE;
	AssemblyMaterialMove : BOOL;
	F_VisionSensor1 	 : F_TRIG;
	F_VisionSensor2 	 : F_TRIG;
	Clamping1 : BOOL;
	Clamping2 : BOOL;
	F_AssemblyExit : F_TRIG;
	AssemblyConvMove : BOOL;
	Clamping3 : BOOL;
	F_AssembledPosition : F_TRIG;
	TwoAxis1Working : BOOL;
END_VAR

IF OPC.iAssemblyStart AND OPC.iAssemblyEmergency AND OPC.iAssemblyStop AND OPC.iAssemblyAutomatic THEN
	Start := TRUE;
ELSE
	Start := FALSE;
END_IF


IF TwoAxis1Working THEN
	Part1Ready := FALSE;
	Part2Ready := FALSE;
END_IF
// At first we want to make CTUD counter which will count how many parts are in move
Counter1(CU := iMachine1Exit, CD:= VisionSensor1);
Counter2(CU := iMachine2Exit, CD:= VisionSensor2);

// Now when we have our counter, if the CV is bigger than 0, QD whille be false so we have mocing part
LiquidMaterialConv1 := NOT Counter2.QD;

// Same as above, if CV bigger than 0, conv should move if possible
BaseMaterialConv1 := NOT Counter1.QD;



(* Two Axis Pick & Place which assemble two parts, two vision sensors, two right positioners and  light conv behind them *)

// At first we want to make falling trigger using vision senser, those numbers are taken from factory i/o
IF iVisionSenserPart1 = 2 OR iVisionSenserPart1 = 5 OR iVisionSenserPart1 = 8 THEN
	VisionSensor1 := TRUE;
ELSE 
	VisionSensor1 := FALSE;
END_IF;

// Same as previous we want to check when expected material went in
IF iVisionSenserPart2 = 3 OR iVisionSenserPart2 = 6 OR iVisionSenserPart2 = 9 THEN
	VisionSensor2 := TRUE;
ELSE 
	VisionSensor2 := FALSE;
END_IF;

// Making falling trigger 
F_VisionSensor1(CLK := VisionSensor1);
F_VisionSensor2(CLK := VisionSensor2);

// Checking if the parts are on positon, then clamping them
IF F_VisionSensor1.Q THEN 
	Clamping1 := TRUE;
END_IF;

// Checking if clamped
IF Clamping1 AND iRightPositioner1Clamped THEN
	Part1Ready := TRUE;
	Clamping1 := FALSE;
END_IF;

// Now the very same thing for second positioner

// Checking if the parts are on positon, then clamping them
IF F_VisionSensor2.Q THEN 
	Clamping2 := TRUE;
END_IF;

// Checking if clamped
IF Clamping2 AND iRightPositioner2Clamped THEN
	Part2Ready := TRUE;
END_IF;

//////////////////
IF TwoAxis1.JobDone THEN
	RaisePositioner2 := TRUE;
	Clamping2 := FALSE; 
END_IF;

// When right positioner is up, move material
IF RaisePositioner2 AND  iRightPositioner1OnPlace THEN
	AssemblyMaterialMove := TRUE;
END_IF;

// Close opened right positioner 2
F_AssemblyExit(CLK := iAtAssembledConvEntry);
IF F_AssemblyExit.Q THEN
	AssemblyMaterialMove := FALSE;
	AssemblyConvMove := TRUE;
	RaisePositioner2 := FALSE;
END_IF;

// Falling trigger at the end of this conv
F_AssembledPosition(CLK := OPC.iAtAssemledPosition);

// When f_trig at the end, stop conveyor
IF F_AssembledPosition.Q THEN
	AssemblyConvMove := FALSE;
	Clamping3 := TRUE;
END_IF;


oEmitter1Emit := HMI.EmittMaterials;
oEmitter1Part := HMI.Emitter1Color;
oRawMaterialSupply1 := NOT iMachine1Entry AND NOT iMachiningCenter1IsBusy;
oMachiningCenter1Start := iMachine1Entry;
oMachiningCenter1Product := TRUE;

oEmitter2Emit := HMI.EmittMaterials;
oEmitter2Part := HMI.Emitter2Color;
oRawMaterialSupply2 := NOT iMachine2Entry AND NOT iMachiningCenter2IsBusy;
oMachiningCenter2Start := iMachine2Entry;
oMachiningCenter2Product := FALSE;

oLiquidMaterialConv1 := NOT TwoAxis1Working AND LiquidMaterialConv1 ;
oLiquidMaterialConv2 := NOT TwoAxis1Working OR AssemblyMaterialMove;

oBaseMaterialConv1 := NOT TwoAxis1Working AND BaseMaterialConv1 ;
oBaseMaterialConv2 := NOT TwoAxis1Working;

oRightPositioner1Clamp := Clamping1;
oRightPositioner1Raise := RaisePositioner2;

oRightPositioner2Clamp := Clamping2;
oRightPositioner2Raise := RaisePositioner2;

oRightPositioner3Clamp := Clamping3;

oAssembledMaterialConv := AssemblyConvMove OR iAtAssembledConvEntry;

END_FUNCTION_BLOCK

// Device/Application/TwoAxisLogic
FUNCTION_BLOCK TwoAxisLogic
VAR_INPUT
	Start   : BOOL;
	Grabbed : BOOL;
	MovingX : BOOL;
	MovingZ : BOOL;
	IncomingArray : ARRAY[0..8] OF INT;
END_VAR
VAR_OUTPUT
	X : BOOL;
	Z : BOOL;
	Grab : BOOL;
	JobDone : BOOL;
END_VAR
VAR
	F_MoveZ : F_TRIG;
	F_MoveX : F_TRIG;
	MyIncrement : INT := 0;
	XX : BOOL := FALSE;
	ZZ : BOOL := FALSE;
END_VAR

F_MoveZ(CLK := MovingZ);
F_MoveX(CLK := MovingX);
IF F_MoveZ.Q THEN
	ZZ := TRUE;
END_IF
IF F_MoveX.Q THEN
	XX := TRUE;
END_IF

IF START THEN
CASE IncomingArray[Myincrement] OF
	0:
		JobDone := TRUE;
	1:
		Z := TRUE;
		IF ZZ AND( MyIncrement = 0 OR MyIncrement = 1 ) AND Grabbed THEN
			Grab := TRUE;
			ZZ := FALSE;
			MyIncrement := MyIncrement + 1;
		ELSIF ZZ AND( MyIncrement = 3 OR MyIncrement = 4 ) THEN
			Grab := FALSE;
			ZZ := FALSE;
			MyIncrement := MyIncrement + 1;
		END_IF;
	2:
		X := TRUE;
		IF  XX THEN
			MyIncrement := MyIncrement + 1;
			XX := FALSE;
		END_IF;
	3:
		Z := FALSE;
		IF ZZ THEN
			MyIncrement := MyIncrement + 1;
			ZZ := FALSE;
		END_IF;
	4:
		X := FALSE;
		IF XX THEN
			MyIncrement := MyIncrement + 1;
			XX := FALSE;
		END_IF;
END_CASE
ELSE
	MyIncrement := 0;
	JobDone := FALSE;
	ZZ := FALSE;
	XX := FALSE;
END_IF;

END_FUNCTION_BLOCK

// Device/Application/Round
FUNCTION Round : REAL
VAR_INPUT
	First : REAL;
END_VAR
VAR
END_VAR

Round := TO_LREAL(TO_DINT(First * 100.0)/100.0);

END_FUNCTION

// Device/Application/Crane
FUNCTION_BLOCK Crane
VAR_INPUT
	LeftOrRight : BOOL; // if pick material from left then 0 if from right then 1
	Swap : BOOL;
	Place : BOOL;
	Pick : BOOL;
	CraneLeftLimit : BOOL;
	CraneRightLimit : BOOL;
	CraneMidLimit : BOOL;
	CraneMovingZ : BOOL;
	CraneMovingX : BOOL;
	CraneAtStart : BOOL;
	WantedMaterial : INT;
	WarehouseNumer : INT;
	CanEnd : BOOL;
END_VAR
VAR_OUTPUT
	CraneTargetPosition : INT := 100;
	CraneRight : BOOL := FALSE; 
	CraneLeft : BOOL := FALSE; 
	CraneLift : BOOL := FALSE; 
	JobDone : BOOL := FALSE; 
	Working : BOOL := FALSE; 
END_VAR
VAR
	Counter : INT := 1;
	F_MovingZ : F_TRIG;
	F_MovingX : F_TRIG;
	MovingZ : BOOL := FALSE;
	MovingX : BOOL := FALSE;
	Pic : BOOL := FALSE;
	Pla : BOOL := FALSE;
	Swa : BOOL := FALSE;
	CraneDesignedLocation : INT;
	ProbablyReady : TON;
END_VAR

IF Place OR Swap AND NOT CraneAtStart AND NOT Working THEN
	CraneTargetPosition  := 100;
	MovingZ := FALSE;
	MovingX := FALSE;
END_IF;
IF Pick AND NOT Working THEN
	Counter := 7;
	Working := TRUE;
	Pic := TRUE;
	MovingZ := FALSE;
	MovingX := FALSE;
ELSIF Place AND NOT Pick AND NOT Working AND ProbablyReady.Q THEN
	Counter := 13;
	Working := TRUE;
	Pla := TRUE;
	MovingZ := FALSE;
	MovingX := FALSE;
ELSIF Swap AND NOT Place AND NOT Pick AND NOT Working AND ProbablyReady.Q  THEN
	Working := TRUE;
	Swa := TRUE;
	Counter := 13;
	MovingZ := FALSE;
	MovingX := FALSE;
END_IF

ProbablyReady(IN := CraneAtStart,PT := T#500MS);
F_MovingX(CLK := CraneMovingX);
F_MovingZ(CLK := CraneMovingZ);
	
// Falling triggers
IF F_MovingX.Q THEN
	MovingX := TRUE;
END_IF;
	
IF F_MovingZ.Q THEN
	MovingZ := TRUE;
END_IF;

CASE Counter OF
	0:
		CraneRight := FALSE;
		CraneLeft := FALSE;
		CraneLift := FALSE;
		JobDone := TRUE;
		CraneTargetPosition := 100;
		Working := FALSE;
		Pla := FALSE;
		Pic := FALSE;
		Swa := FALSE;
		MovingZ := FALSE;
		MovingX := FALSE;
	7:
		IF Pla THEN
			CraneDesignedLocation := FindFreePlace(WarehouseNumer);
		ELSIF Pic THEN
			CraneDesignedLocation := WhereIsMaterial(WarehouseNumer := WarehouseNumer, WantedMaterial := WantedMaterial);
		END_IF
		CraneTargetPosition := CraneDesignedLocation;
		IF (MovingZ AND MovingX) OR (MovingX AND CraneTargetPosition < 10) THEN
			Counter := 14;
			MovingZ := FALSE;
			MovingX := FALSE;
		END_IF	
	8:
		CraneTargetPosition := 100;
		IF (MovingZ AND MovingX) OR (MovingX AND CraneTargetPosition < 10) AND NOT CanEnd THEN
			Counter := 12;
			MovingZ := FALSE;
			MovingX := FALSE;
		END_IF
	12: 
		CraneLeft := NOT MovingZ AND LeftOrRight;
		CraneRight := NOT MovingZ AND NOT LeftOrRight;
		IF CraneRightLimit OR CraneLeftLimit THEN
			CraneLift := FALSE;
		END_IF
		IF MovingZ AND CraneMidLimit THEN
			MovingZ := FALSE;
			Counter := 0;
		END_IF
	13:
		CraneLeft := NOT CraneLift AND NOT LeftOrRight;
		CraneRight := NOT CraneLift AND LeftOrRight;
		IF CraneRightLimit OR CraneLeftLimit THEN
			CraneLift := TRUE;
		END_IF
		IF MovingZ AND CraneMidLimit AND NOT swa THEN
			MovingZ := FALSE;
			MovingX := FALSE;
			Counter := 7;
		ELSIF MovingZ AND CraneMidLimit AND swa AND NOT CanEnd THEN
			MovingZ := FALSE;
			MovingX := FALSE;
			Counter := 12;
		END_IF
	14:	
		CraneRight := NOT MovingZ;
		IF CraneRightLimit AND Pla THEN
			CraneLift := FALSE;
			FillWarehouseArray(Place := CraneTargetPosition, ZeroOrOne := TRUE, WarehouseNumer := WarehouseNumer );
			// Here also add the info what we store
		ELSIF CraneRightLimit AND Pic THEN
			CraneLift := TRUE;
			FillWarehouseArray(Place := CraneTargetPosition, ZeroOrOne := FALSE, WarehouseNumer := WarehouseNumer );
		END_IF
		IF MovingZ AND CraneMidLimit AND Pla THEN
			MovingZ := FALSE;
			MovingX := FALSE;
			IF Pick THEN
				Pla := FALSE;
				Pic := TRUE;
				Counter := 7;
			ELSE
				Counter := 0;
			END_IF
		ELSIF MovingZ AND CraneMidLimit AND Pic THEN
			MovingZ := FALSE;
			MovingX := FALSE;
			Counter := 8;
		END_IF
END_CASE

END_FUNCTION_BLOCK

// Device/Application/FindFreePlace
FUNCTION FindFreePlace : INT
VAR_INPUT
	WarehouseNumer : INT;
END_VAR
VAR
	I : INT;
	J : INT := 0;
END_VAR

IF WarehouseNumer = 1 THEN
	J := 0;
	FOR I:=1 TO 54 DO 
	   IF GVL.Warehouse1Array[I] = 0 THEN
	   	  J:=I; 
	      EXIT; 
	   END_IF;
	END_FOR;
ELSIF WarehouseNumer = 2 THEN
	J := 0;
	FOR I:=1 TO 54 DO 
	   IF GVL.Warehouse2Array[I] = 0 THEN
	   	  J:=I; 
	      EXIT; 
	   END_IF;
	END_FOR;
END_IF
FindFreePlace := J;

END_FUNCTION

// Device/Application/WhereIsMaterial
FUNCTION WhereIsMaterial : INT
VAR_INPUT
	WantedMaterial : INT;
	WarehouseNumer : INT;
END_VAR
VAR
	I : INT;
	J : INT := 0;
END_VAR

IF WarehouseNumer = 1 THEN
J := 0;
FOR I:=1 TO 54 DO 
   IF GVL.Warehouse1ArrayMaterial[I] = WantedMaterial THEN
   	  J:=I; 
      EXIT; 
   END_IF;
END_FOR;
ELSIF WarehouseNumer = 2 THEN
J := 0;
FOR I:=1 TO 54 DO 
   IF GVL.Warehouse2ArrayMaterial[I] = WantedMaterial THEN
   	  J:=I; 
      EXIT; 
   END_IF;
END_FOR;
	
END_IF
WhereIsMaterial := J;

END_FUNCTION

// Device/Application/FillWarehouseArray
FUNCTION FillWarehouseArray : INT
VAR_INPUT
	Place : INT;
	ZeroOrOne : BOOL;
	WarehouseNumer : INT;
END_VAR
VAR
END_VAR

IF WarehouseNumer = 1 THEN
	IF ZeroOrOne THEN
		GVL.Warehouse1Array[Place] := 1;
	ELSE
		GVL.Warehouse1Array[Place] := 0;
		HMI.Pick1 := FALSE;
		HMI.WantedMaterial1 := 0;	
	END_IF
ELSIF WarehouseNumer = 2 THEN
	IF ZeroOrOne THEN
		GVL.Warehouse2Array[Place] := 1;
	ELSE
		GVL.Warehouse2Array[Place] := 0;	
		HMI.Pick2 := FALSE;
		HMI.WantedMaterial2 := 0;	
	END_IF
END_IF

END_FUNCTION

// Device/Application/ExitMagazine
FUNCTION_BLOCK ExitMagazine
VAR_INPUT
	iAtCrane1Exit : BOOL;
	iAtCrane2Exit : BOOL;
	iAtTurntable2Entry : BOOL;
	iAtTurntable2Exit : BOOL;
	iAtTurntable2ExitWarehouse1 : BOOL;
	iAtTurntable2ExitWarehouse2 : BOOL;
	iAtExitWarehouseExit : BOOL;
	iTurntable2Back : BOOL;
	iTurntable2Front : BOOL;
	iTurntable2Atzero : BOOL;
	iTurntable2AtNinety : BOOL;
END_VAR
VAR_OUTPUT
	oExitWarehouseConv1 : BOOL;
	oExitWarehouseConv2 : BOOL;
	oFirstWarehouseConvLoadOpposite : BOOL;
	oSecondWarehouseLoadConvOpposite : BOOL;
	oTowardSecondWarehouse : BOOL;
	oTurntable2Turn : BOOL;
	oTurntable2Forward : BOOL;
	oTurntable2Backward : BOOL;
END_VAR
VAR
	R_Crane1 : R_TRIG;
	R_Crane2 : R_TRIG;
	F_TurnLeft : F_TRIG;
	F_TurnRight : F_TRIG;
	R_TurnFrontStop : R_TRIG;
	R_TurnBackStop : R_TRIG;
	F_TurnLeave : F_TRIG;
	F_ConvLeave : F_TRIG;
	F_ConvLeave1 : F_TRIG;
	Conv1Left : BOOL;
	Conv1Right : BOOL;
	Conv1Exit : BOOL;
	Conv2Exit : BOOL;
	EntryLeft : BOOL;
	EntryRight : BOOL;
	TurnForward : BOOL;
	TurnBackward : BOOL;
	TurnBusy : BOOL;
END_VAR

R_Crane1(CLK := iAtCrane1Exit);
R_Crane2(CLK := iAtCrane2Exit);

IF R_Crane1.Q THEN
	Conv1Left := TRUE;
END_IF

IF R_Crane2.Q THEN
	Conv1Right := TRUE;
END_IF

IF iAtTurntable2Entry AND NOT TurnBusy AND NOT EntryRight AND NOT oSecondWarehouseLoadConvOpposite THEN
	EntryLeft := TRUE;
END_IF

IF iAtTurntable2Exit AND NOT TurnBusy AND NOT EntryLeft THEN
	EntryRight := TRUE;
END_IF

F_TurnLeft(CLK := iAtTurntable2Entry);
F_TurnRight(CLK := iAtTurntable2Exit);

IF F_TurnLeft.Q THEN
	Conv1Left := FALSE;
	TurnForward := TRUE;
END_IF

IF F_TurnRight.Q THEN
	Conv1Right := FALSE;
	TurnBackward := TRUE;
END_IF

R_TurnFrontStop(CLK := iTurntable2Front);
R_TurnBackStop(CLK := iTurntable2Back);

IF R_TurnFrontStop.Q AND TurnForward THEN
	TurnForward := FALSE;
	oTurntable2Turn := TRUE;
	TurnBusy := TRUE;
	EntryLeft := FALSE;
ELSIF R_TurnBackStop.Q AND TurnBackward THEN
	TurnBackward := FALSE;
	oTurntable2Turn := TRUE;
	TurnBusy := TRUE;
	EntryRight := FALSE;
END_IF

IF iTurntable2AtNinety THEN
	TurnForward := TRUE;
	Conv1Exit := TRUE;
END_IF

F_TurnLeave( CLK := iAtTurntable2ExitWarehouse1);

IF F_TurnLeave.Q THEN
	TurnForward := FALSE;
	oTurntable2Turn := FALSE;
END_IF

IF TurnBusy AND iTurntable2Atzero AND (NOT iTurntable2Front AND NOT iTurntable2Back)  THEN
	TurnBusy := FALSE;
END_IF

F_ConvLeave1(CLK:= iAtTurntable2ExitWarehouse2);
IF F_ConvLeave1.Q THEN
	Conv1Exit := FALSE;
	Conv2Exit := TRUE;
END_IF

F_ConvLeave(CLK:= iAtExitWarehouseExit);
IF F_ConvLeave.Q THEN
	Conv2Exit := FALSE;
END_IF

	oExitWarehouseConv1 := Conv1Exit OR iAtTurntable2ExitWarehouse1;
	oExitWarehouseConv2 := Conv2Exit OR iAtTurntable2ExitWarehouse2;
	oFirstWarehouseConvLoadOpposite := Conv1Left;
	oSecondWarehouseLoadConvOpposite := Conv1Right AND (NOT TurnBusy OR NOT iAtTurntable2Exit) AND NOT EntryLeft;
	oTowardSecondWarehouse := Conv1Left AND (NOT TurnBusy OR NOT iAtTurntable2Entry) AND NOT EntryRight;
	oTurntable2Forward := EntryLeft OR TurnForward; 
	oTurntable2Backward := EntryRight OR TurnBackward;

END_FUNCTION_BLOCK

// Device/Application/ThreeAxis
FUNCTION_BLOCK ThreeAxis
VAR_INPUT
	iBoxSupplyStart : BOOL;
	iBoxSupplyStop : BOOL;
	iSafetyDoorBoxSupply : BOOL;
	iBigBox : BOOL;
	iMidBox : BOOL;
	iSmallBox : BOOL;
	iAtBoxSupplyEnter : BOOL;
	iAtBoxSupplyCurveConv2Entry : BOOL;
	iAtBoxSupplyCurveConv2Exit : BOOL;
	iAtPalletDestinationEntry : BOOL;
	iAtPalletDestinationExit : BOOL;
	iAtLoadEmptyBoxEntry : BOOL;
	iAtLoadEmptyBoxExit : BOOL;
	iAtSecondWarehouseCurveConv3Entry : BOOL;
	iPickPlace1Rotated : BOOL;
	iPickPlace1CurrentX : REAL;
	iPickPlace1CurrentY : REAL;
	iPickPlace1CurrentZ : REAL;
	iPickPlace1BoxDetected : BOOL;
	iAtSecondWarehouseCurveConv3Exit : BOOL;
	iAtElevatorEntry : BOOL;
	iElevator1CurrentPoint : REAL;
	iAtSecondWarehouseConv5 : BOOL;
	ElevatorBusy : BOOL;
END_VAR
VAR_OUTPUT
	oBoxSupplyConv1 : BOOL;
	oBoxSupplyConv3 : BOOL;
	oBoxSupplyCurveConv2 : BOOL;
	oEmptyBoxConvSupply : BOOL;
	oPickPlace1X : REAL;
	oPickPlace1Y : REAL;
	oPickPlace1Z : REAL;
	oPickPlace1Grab : BOOL;
	oSecondWarehouseConv1 : BOOL;
	oSecondWarehouseConv12 : BOOL;
	oSecondWarehouseConv2 : BOOL;
	oSecondWarehouseCurveConv3 : BOOL;
	oSecondWarehouseConv4 : BOOL;
	oSecondWarehouseConv5 : BOOL;
END_VAR
VAR
	BoxSupplyStart : BOOL;
	CanFinish : BOOL;
	JobDone: BOOL;
	LegitProductArray : ARRAY[0..30] OF BOOL;
	EntryPointer : INT := 0;
	ExitPointer : INT := 0;
	F_BoxMeasure : F_TRIG;
	R_CurveConvEntry : R_TRIG;
	R_CurveConvExit : R_TRIG;
	F_DestinationEntry : F_TRIG;
	F_DestinationExit : F_TRIG;
	F_Reload : F_TRIG;
	F_PickPlaceLeave : F_TRIG;
	F_LastPart : F_TRIG;
	F_LongStraight : F_TRIG;
	F_End : F_TRIG;
	F_FirstCurveExit : F_TRIG;
	F_LastConv : F_TRIG;
	BoxPlaced : CTU;
	PickPlaceWorking : BOOL;
	PalleteOnPlace : BOOL;
	BoxOnPlace : BOOL := FALSE;
	SwitchCase : INT := 30;
	X : REAL;
	Y : REAL;
	Conv3 : BOOL;
	Conv2 : BOOL;
	Conv12 : BOOL;
	Conv13 : BOOL;
	Conv14 : BOOL;
	Conv15 : BOOL;
	Conv16 : BOOL;
	RealX : REAL;
	RealZ : REAL;
	RealY : REAL;
	RealE : REAL;
	Finished : BOOL;
	WaitForGrab : TON;
	Grab : BOOL;
END_VAR

IF iBoxSupplyStart AND iBoxSupplyStop THEN
	BoxSupplyStart := TRUE;
ELSIF NOT iBoxSupplyStop THEN
	BoxSupplyStart := FALSE;
END_IF
IF BoxSupplyStart THEN
	F_BoxMeasure(CLK := iAtBoxSupplyEnter);
	IF F_BoxMeasure.Q THEN
		IF iBigBox AND iMidBox AND iSmallBox THEN
			LegitProductArray[EntryPointer] := 1;
			EntryPointer := EntryPointer + 1;
			IF EntryPointer > 30 THEN
				EntryPointer := 0;
			END_IF 
		ELSIF NOT iBigBox AND ((iMidBox AND iSmallBox) OR iSmallBox) THEN
			LegitProductArray[EntryPointer] := 0;
			EntryPointer := EntryPointer + 1;
			IF EntryPointer > 30 THEN
				EntryPointer := 0;
			END_IF 
		END_IF
	END_IF

	R_CurveConvEntry(CLK := iAtBoxSupplyCurveConv2Entry);
	IF R_CurveConvEntry.Q THEN
		Conv2 := TRUE;
	END_IF

	F_FirstCurveExit(CLK := iAtBoxSupplyCurveConv2Exit);
	IF F_FirstCurveExit.Q THEN
		Conv2 := FALSE;
	END_IF
	
	R_CurveConvExit(CLK := iAtBoxSupplyCurveConv2Exit);
	IF R_CurveConvExit.Q THEN
		Conv3 := TRUE;
	END_IF
	
	//oBoxSupplyConv1 := NOT iAtBoxSupplyCurveConv2Entry OR NOT BoxOnPlace;
	oBoxSupplyConv1 := NOT BoxOnPlace;
	oBoxSupplyConv3 :=  NOT BoxOnPlace;
	oBoxSupplyCurveConv2 :=  NOT BoxOnPlace;
	//oBoxSupplyCurveConv2 := Conv2 AND (NOT iAtBoxSupplyCurveConv2Exit OR NOT BoxOnPlace);
	//oBoxSupplyCurveConv2 := (Conv2 AND(NOT iAtBoxSupplyCurveConv2Exit OR NOT BoxOnPlace)) OR (iAtBoxSupplyCurveConv2Exit AND NOT BoxOnPlace);
	oEmptyBoxConvSupply := NOT PalleteOnPlace;
	oSecondWarehouseConv12 := (Conv12 AND (CanFinish OR NOT iAtLoadEmptyBoxExit));
	oSecondWarehouseConv1 := NOT PalleteOnPlace;
	oSecondWarehouseConv2 := ( Conv13 AND (CanFinish OR NOT iAtSecondWarehouseCurveConv3Entry));
	oSecondWarehouseCurveConv3 := Conv14 AND (CanFinish OR NOT iAtSecondWarehouseCurveConv3Exit);
	oSecondWarehouseConv4 := Conv15 AND (CanFinish OR NOT iAtSecondWarehouseConv5);
	oSecondWarehouseConv5 := Conv16 AND (CanFinish OR NOT iAtElevatorEntry) AND NOT ElevatorBusy;
	
	F_DestinationEntry(CLK := iAtPalletDestinationEntry);
	IF F_DestinationEntry.Q THEN
		IF LegitProductArray[ExitPointer] = 1 THEN
			BoxOnPlace := TRUE;
			ExitPointer := ExitPointer + 1;
			IF ExitPointer > 30 THEN
				ExitPointer := 0;
			END_IF
		ELSE
			ExitPointer := ExitPointer + 1;
		END_IF
	END_IF
	F_Reload(CLK := iAtLoadEmptyBoxEntry);
	IF F_Reload.Q THEN
		PalleteOnPlace := TRUE;
	END_IF

	IF BoxOnPlace AND PalleteOnPlace AND NOT PickPlaceWorking THEN
		PickPlaceWorking := TRUE;
		SwitchCase := 1;
	END_IF

	IF JobDone THEN
		BoxOnPlace := FALSE;
		PickPlaceWorking := FALSE;
		JobDone := FALSE;
		Finished := TRUE;
	END_IF

	BoxPlaced(CU := Finished, PV := 4); 
	IF BoxPlaced.Q THEN
		BoxPlaced.RESET := TRUE;
		PalleteOnPlace := FALSE;
		Conv12 := TRUE;
	END_IF
	
	IF iAtLoadEmptyBoxExit THEN
		Conv13 := TRUE;
	END_IF
	
	F_PickPlaceLeave(CLK := iAtLoadEmptyBoxExit);
	IF F_PickPlaceLeave.Q THEN
		Conv12 := FALSE;
	END_IF
	
	IF iAtSecondWarehouseCurveConv3Entry THEN
		Conv14 := TRUE;
	END_IF

	F_LastPart(CLK := iAtSecondWarehouseCurveConv3Entry);
	IF F_LastPart.Q THEN
		Conv13 := FALSE;
	END_IF

	IF iAtSecondWarehouseCurveConv3Exit THEN
		Conv15 := TRUE;
	END_IF
	
	F_LongStraight(CLK := iAtSecondWarehouseCurveConv3Exit);
	IF F_LongStraight.Q THEN
		Conv14 := FALSE;
	END_IF
	
	IF iAtSecondWarehouseConv5 THEN
		Conv16 := TRUE;
	END_IF
	F_LastConv(CLK := iAtSecondWarehouseConv5);
	IF F_LastConv.Q THEN
		Conv15 := FALSE;
	END_IF
	
	F_End(CLK := iAtElevatorEntry);
	IF F_End.Q THEN
		Conv16 := FALSE;
	END_IF
	
	RealE := Round(First := iElevator1CurrentPoint);
	
	IF RealE = 0.0 THEN
		CanFinish := TRUE;
	ELSE
		CanFinish := FALSE;
	END_IF
	
	WaitForGrab(IN := Grab, PT := T#500MS);
	
	RealX := Round(First := iPickPlace1CurrentX);
	RealZ := Round(First := iPickPlace1CurrentZ);
	RealY := Round(First := iPickPlace1CurrentY);
	
	IF PickPlaceWorking THEN
		CASE SwitchCase OF
			0:
				oPickPlace1X := 1.5; 
				oPickPlace1Y := 4.5; 
				oPickPlace1Z := 0.0; 
				JobDone := TRUE;
			1:
				Finished := FALSE;
				BoxPlaced.RESET := FALSE;
				oPickPlace1X := 1.5; 
				oPickPlace1Y := 4.5; 
				oPickPlace1Z := 0.0; 
				IF RealX = oPickPlace1X AND RealY = oPickPlace1Y  AND RealZ = oPickPlace1Z THEN
					SwitchCase := 2;
				END_IF
			2:
				oPickPlace1Z := 7.8;
				IF RealZ = oPickPlace1Z THEN
					Grab := TRUE;
					oPickPlace1Grab := TRUE;
				END_IF
				IF WaitForGrab.Q THEN
					Grab := FALSE;
					SwitchCase := 3;
				END_IF 
			3: 
				oPickPlace1Z := 0.0; 
				IF RealZ = oPickPlace1Z THEN
					SwitchCase := 4;
				END_IF
			4:
				IF BoxPlaced.CV = 0.0 THEN
					oPickPlace1X := 6.5; 
					oPickPlace1Y := 6.0; 
				ELSIF BoxPlaced.CV = 1 THEN
					oPickPlace1X := 8.3; 
					oPickPlace1Y := 6.0;
				ELSIF BoxPlaced.CV = 2 THEN
					oPickPlace1X := 6.5; 
					oPickPlace1Y := 9.0; 
				ELSIF BoxPlaced.CV = 3 THEN
					oPickPlace1X := 8.3; 
					oPickPlace1Y := 9.0; 
				END_IF
				IF RealX = oPickPlace1X AND RealY = oPickPlace1Y THEN
					SwitchCase := 5;
				END_IF
			5:
				oPickPlace1Z := 7.8; 
				IF RealZ = oPickPlace1Z THEN
					oPickPlace1Grab := FALSE;
					SwitchCase := 6;
				END_IF
			6:
				oPickPlace1Z := 0.0; 
				IF RealZ = oPickPlace1Z THEN
					SwitchCase := 0;
				END_IF
		END_CASE
	END_IF
END_IF

END_FUNCTION_BLOCK

// Device/Application/PalletizerElevator
FUNCTION_BLOCK PalletizerElevator
VAR_INPUT
	iPalletizerAutomatic : BOOL;
	iPalletizerManual : BOOL;
	iPalletizerEmergency : BOOL;
	iPalletizerStart : BOOL;
	iPalletizerStop : BOOL;
	iAtElevatorUpEntry : BOOL; 
	iAtElevatorExit : BOOL; 
	iAtElevatorEntry : BOOL; 
	iElevator1RightLimit : BOOL; 
	iElevator1LeftLimit : BOOL; 
	iElevator1CurrentPoint  : REAL;
	iPalletizer1ElevatorMoving : BOOL; 
	iAtPalletizerConvEntry : BOOL; 
	iAtPalletizerChainEntry : BOOL; 
	iPalletizer1ElevatorBack : BOOL; 
	iPalletizer1ElevatorFront : BOOL; 
	iAtPalletizerEntry : BOOL; 
	iPalletizer1Opening : BOOL; 
	iPalletizer1Clamped : BOOL; 
	iPalletizer1Pushing : BOOL; 
END_VAR
VAR_OUTPUT
	oElevator1Forward : BOOL;
	oElevator1SetPoint : REAL;
	oPalletizer1Open : BOOL := FALSE;
	oPalletizer1Push : BOOL;
	oPalletizer1Clamp : BOOL;
	oPalletizer1Forward : BOOL;
	oPalletizer1ElevatorUp : BOOL;
	oPalletizer1ChainForward : BOOL;
	oPalletizer1ElevatorDown : BOOL;
	oPalletizer1ChainBackward : BOOL;
	oPalletizer1ElevatorMoveToMax : BOOL;
	oPalletizerConv : BOOL;
	oPalletizerSupplyConv : BOOL;
	oPalletizerSupplyLightConv : BOOL;
	oPalletsTowardElevator : BOOL;
	oPalletizer1Turn : BOOL;
	ElevatorBusy : BOOL;
END_VAR
VAR
	Stop : BOOL;
	SetHigh : REAL;
	PalletizerStart : BOOL := FALSE;
	R_Pushing : F_TRIG;
	F_RightLimit : F_TRIG;
	Direction : BOOL := FALSE;
	F_EntryLightConv : F_TRIG;
	ThreeOnTwo : INT := 0;
	TwoOnThree : INT := 0;
	ThreeRounds : INT := 0;
	TwoRounds : INT := 0;
	PalletizerElevator : BOOL := FALSE;
	InElevator : BOOL := FALSE;
	F_PalletizerChain : F_TRIG;
	F_MovingPalletizerElevator : F_TRIG;
	MovingZ : BOOL := FALSE;
	PalleteReady : BOOL := FALSE;
	F_Push : F_TRIG;
	MoveDown : BOOL := FALSE;
	Layers : CTU;
	F_EnterLow : F_TRIG;
	F_EnterElevator : F_TRIG;
	F_AlmostWarehouse : F_TRIG;
	ElevatorUp : BOOL := FALSE;
	ElevatorDown : BOOL := FALSE;
	ElvatorTakingUp : BOOL := FALSE;
	ElvatorTakingDown : BOOL := FALSE;
	Pushed : BOOL := FALSE;
	NotiPalletizer1Pushing : BOOL := FALSE;
	SwitchCase : INT := 30;
	ShutDown : BOOL := FALSE;
	PickUp : BOOL := FALSE;
	Throw : BOOL := FALSE;
	TimeUp : TON;
	Busy : BOOL;
END_VAR

IF iPalletizerStart AND iPalletizerStop AND iPalletizerEmergency THEN
	PalletizerStart := TRUE;
	SwitchCase := 1;
ELSIF NOT iPalletizerStop AND iPalletizerEmergency THEN
	Stop := TRUE;
ELSIF NOT iPalletizerEmergency THEN
	SwitchCase := 0;
END_IF

GVL.PalletizerArray[9] := NOT PalletizerElevator; //  oPalletizerSupplyConv
GVL.PalletizerArray[10] := NOT PalletizerElevator; //  oPalletizerConv
GVL.PalletizerArray[11] := NOT PalletizerElevator;; //  oPalletizer1ChainForward

ElevatorUp := Round(First := iElevator1CurrentPoint) = 4.65;
ElevatorDown := Round(First := iElevator1CurrentPoint) = 0.0;

F_AlmostWarehouse(CLK := iAtElevatorExit);

F_PalletizerChain(CLK := iAtPalletizerChainEntry);
IF F_PalletizerChain.Q THEN
	InElevator := TRUE;
END_IF
	
F_MovingPalletizerElevator(CLK :=iPalletizer1ElevatorMoving);
IF F_MovingPalletizerElevator.Q THEN
	MovingZ := TRUE;
END_IF
	
IF InElevator AND iPalletizer1ElevatorBack AND iPalletizer1ElevatorFront THEN
	PalletizerElevator := TRUE;
	InElevator := FALSE;
END_IF

////
IF PalletizerElevator AND NOT PalleteReady THEN
	GVL.PalletizerArray[6] := 1; //  oPalletizer1ElevatorMoveToMax
	GVL.PalletizerArray[7] := 1; //  oPalletizer1ElevatorUp
	IF MovingZ THEN
		GVL.PalletizerArray[6] := 0; //  oPalletizer1ElevatorMoveToMax
		GVL.PalletizerArray[7] := 0; //  oPalletizer1ElevatorUp
		MovingZ := FALSE;
		PalleteReady := TRUE;
	END_IF
END_IF

F_EntryLightConv(CLK := iAtPalletizerEntry);
IF F_EntryLightConv.Q AND Direction THEN
	ThreeOnTwo := ThreeOnTwo + 1;
ELSIF F_EntryLightConv.Q AND NOT Direction THEN
	TwoOnThree := TwoOnThree + 1;
END_IF
	
NotiPalletizer1Pushing := NOT iPalletizer1Pushing;
F_Push(CLK := NotiPalletizer1Pushing);
IF F_Push.Q THEN
	Pushed := TRUE;
END_IF

TimeUp(IN := oPalletizer1Open, PT := T#2000MS);

CASE SwitchCase OF
	0: // Shutdown
		IF NOT ShutDown THEN
			PalletizerStart := FALSE;
			SetArrayToZero();
			ShutDown := TRUE;
		END_IF
	
	1: // Normal working
		ShutDown := FALSE;
		GVL.PalletizerArray[0] := NOT (TwoOnThree = 2 OR ThreeOnTwo = 3) OR NOT iAtPalletizerEntry; // oPalletizerSupplyLightConv
		GVL.PalletizerArray[1] := NOT (TwoOnThree = 2 OR ThreeOnTwo = 3) OR NOT iAtPalletizerEntry; // oPalletizer1Forward
		IF (TwoOnThree = 2 OR ThreeOnTwo = 3) AND iAtPalletizerEntry AND iPalletizer1Opening AND NOT oPalletizer1Open THEN
			SwitchCase := 2;
			TwoOnThree := 0;
			ThreeOnTwo := 0;
		END_IF
	2: // Push
		GVL.PalletizerArray[0] := 0; // oPalletizerSupplyLightConv
		GVL.PalletizerArray[1] := 0; // oPalletizer1Forward
		GVL.PalletizerArray[2] := 1; // oPalletizer1Push
		IF Pushed AND iPalletizer1Pushing THEN
			Pushed := FALSE;
			SwitchCase := 3;
		END_IF
	3: // Back
		GVL.PalletizerArray[2] := 0; // oPalletizer1Push
		IF Pushed AND iPalletizer1Pushing THEN
			Pushed := FALSE;
			IF NOT Direction THEN
					ThreeRounds := ThreeRounds + 1;
			ELSIF Direction THEN
					TwoRounds := TwoRounds + 1;
			END_IF
			IF ThreeRounds = 3 OR TwoRounds = 2 THEN
				Direction := NOT Direction;
				ThreeRounds := 0;
				TwoRounds := 0;
				SwitchCase := 4;
			ELSE
				SwitchCase := 1;
			END_IF
		END_IF
	4:
		GVL.PalletizerArray[3] := 1; //  oPalletizer1Clamp
		IF iPalletizer1Clamped AND PalleteReady THEN
			SwitchCase := 5;
		END_IF
	5:
		GVL.PalletizerArray[4] := 1; //  oPalletizer1Open
		IF TimeUp.Q THEN
			GVL.PalletizerArray[3] := 0; //  oPalletizer1Clamp
			SwitchCase := 6;
		END_IF
	6:
		MoveDown := TRUE;
		GVL.PalletizerArray[5] := 1; //  oPalletizer1ElevatorDown
		IF MovingZ AND NOT Layers.Q THEN
			MovingZ := FALSE;
			MoveDown := FALSE;
			GVL.PalletizerArray[5] := 0; //  oPalletizer1ElevatorDown
			GVL.PalletizerArray[4] := 0; //  oPalletizer1Open
			SwitchCase := 1;
		ELSIF MovingZ AND Layers.Q THEN
			GVL.PalletizerArray[4] := 0; //  oPalletizer1Open
			Layers.RESET := TRUE;
			MovingZ := FALSE;
			MoveDown := FALSE;
			SwitchCase := 7;
		END_IF
	7:
		Layers.RESET := FALSE;
		GVL.PalletizerArray[5] := 1; //  oPalletizer1ElevatorDown
		GVL.PalletizerArray[6] := 1; //  oPalletizer1ElevatorMoveToMax
		IF MovingZ THEN
			GVL.PalletizerArray[5] := 0; //  oPalletizer1ElevatorDown
			GVL.PalletizerArray[6] := 0; //  oPalletizer1ElevatorMoveToMax
			PalleteReady := FALSE;
			PalletizerElevator := FALSE;
			GVL.PalletizerArray[8] := 1; //  oPalletsTowardElevator
			IF Stop THEN
				SwitchCase := 0;
				Stop := FALSE;
			ELSE
				SwitchCase := 1;
			END_IF
			MovingZ := FALSE;
		END_IF
END_CASE

Layers(Cu := MoveDown, PV := 3);

IF iAtElevatorUpEntry AND NOT iAtElevatorEntry AND NOT ElvatorTakingDown THEN
	SetHigh := 4.65;
	ElvatorTakingUp := TRUE;
ELSIF iAtElevatorEntry AND NOT ElvatorTakingUp THEN
	SetHigh := 0.0;
	ElvatorTakingDown := TRUE;
END_IF

IF ElvatorTakingDown AND ElevatorDown THEN
	GVL.PalletizerArray[12] := 1; //  oElevator1Forward
END_IF

IF ElvatorTakingUp AND ElevatorUp AND NOT Throw THEN
	PickUp := TRUE;
	SetHigh := 4.65;
	GVL.PalletizerArray[12] := PickUp ; //  oElevator1Forward
	IF F_RightLimit.Q THEN
		GVL.PalletizerArray[8] := 0; //  oPalletsTowardElevator
		GVL.PalletizerArray[12] := 0 ; //  oElevator1Forward
		SetHigh := 0.0;
		PickUp := FALSE;
		Throw := TRUE;
	END_IF
END_IF

IF Throw AND ElevatorDown THEN
	GVL.PalletizerArray[12] := 1; //  oElevator1Forward
END_IF

IF F_AlmostWarehouse.Q THEN
	ElvatorTakingDown := FALSE;
	ElvatorTakingUp := FALSE;
	Busy := FALSE;
	GVL.PalletizerArray[12] := 0 ; //  oElevator1Forward
	Throw := FALSE;
END_IF

F_RightLimit(CLK:= iElevator1RightLimit);
F_EnterLow(CLK := iAtElevatorEntry);
IF F_RightLimit.Q OR F_EnterLow.Q THEN
	Busy := TRUE;
END_IF

ElevatorBusy := Busy;
oElevator1Forward := (GVL.PalletizerArray[12] AND iPalletizerAutomatic) OR (HMI.oElevator1Forward AND iPalletizerManual);
oElevator1SetPoint := SetHigh;
oPalletizer1Open := (GVL.PalletizerArray[4] AND PalletizerStart AND iPalletizerAutomatic) OR (HMI.oPalletizer1Open AND iPalletizerManual);
oPalletizer1Push := (GVL.PalletizerArray[2] AND (PalletizerStart OR OPC.iAssemblyManual) AND iPalletizerAutomatic) OR (HMI.oPalletizer1Push AND iPalletizerManual);
oPalletizer1Clamp := (GVL.PalletizerArray[3] AND PalletizerStart AND iPalletizerAutomatic) OR (HMI.oPalletizer1Clamp AND iPalletizerManual);
oPalletizer1Forward := (GVL.PalletizerArray[1] AND PalletizerStart AND iPalletizerAutomatic) OR (HMI.oPalletizer1Forward AND iPalletizerManual);
oPalletizer1ElevatorUp := (GVL.PalletizerArray[7] AND PalletizerStart AND iPalletizerAutomatic) OR (HMI.oPalletizer1ElevatorUp AND iPalletizerManual);
oPalletizer1ChainForward := (GVL.PalletizerArray[11] AND PalletizerStart AND iPalletizerAutomatic) OR (HMI.oPalletizer1ChainForward AND iPalletizerManual);
oPalletizer1ElevatorDown := (GVL.PalletizerArray[5] AND PalletizerStart AND iPalletizerAutomatic) OR (HMI.oPalletizer1ElevatorDown AND iPalletizerManual);
oPalletizer1ElevatorMoveToMax := (GVL.PalletizerArray[6] AND PalletizerStart AND iPalletizerAutomatic) OR (HMI.oPalletizer1ElevatorMoveToMax AND iPalletizerManual);
oPalletizerConv := (GVL.PalletizerArray[10] AND PalletizerStart AND iPalletizerAutomatic) OR (HMI.oPalletizerConv AND iPalletizerManual);
oPalletizerSupplyConv := (GVL.PalletizerArray[9] AND PalletizerStart AND iPalletizerAutomatic) OR (HMI.oPalletizerSupplyConv AND iPalletizerManual);
oPalletizerSupplyLightConv := (GVL.PalletizerArray[0] AND PalletizerStart AND iPalletizerAutomatic) OR (HMI.oPalletizerSupplyLightConv AND iPalletizerManual);
oPalletsTowardElevator := ((GVL.PalletizerArray[8] AND (PickUp OR NOT iAtElevatorUpEntry)) AND PalletizerStart AND iPalletizerAutomatic) OR (HMI.oPalletsTowardElevator AND iPalletizerManual);
oPalletizer1Turn := (Direction  AND PalletizerStart AND iPalletizerAutomatic) OR (HMI.oPalletizer1Turn AND iPalletizerManual);

END_FUNCTION_BLOCK

// Device/Application/SetArrayToZero
FUNCTION SetArrayToZero : BOOL
VAR_INPUT
END_VAR
VAR
	I : INT := 0;
END_VAR

FOR I := 0 TO 12 BY 1 DO
	GVL.PalletizerArray[I] := 0;
END_FOR

END_FUNCTION

// Device/Application/Assembly
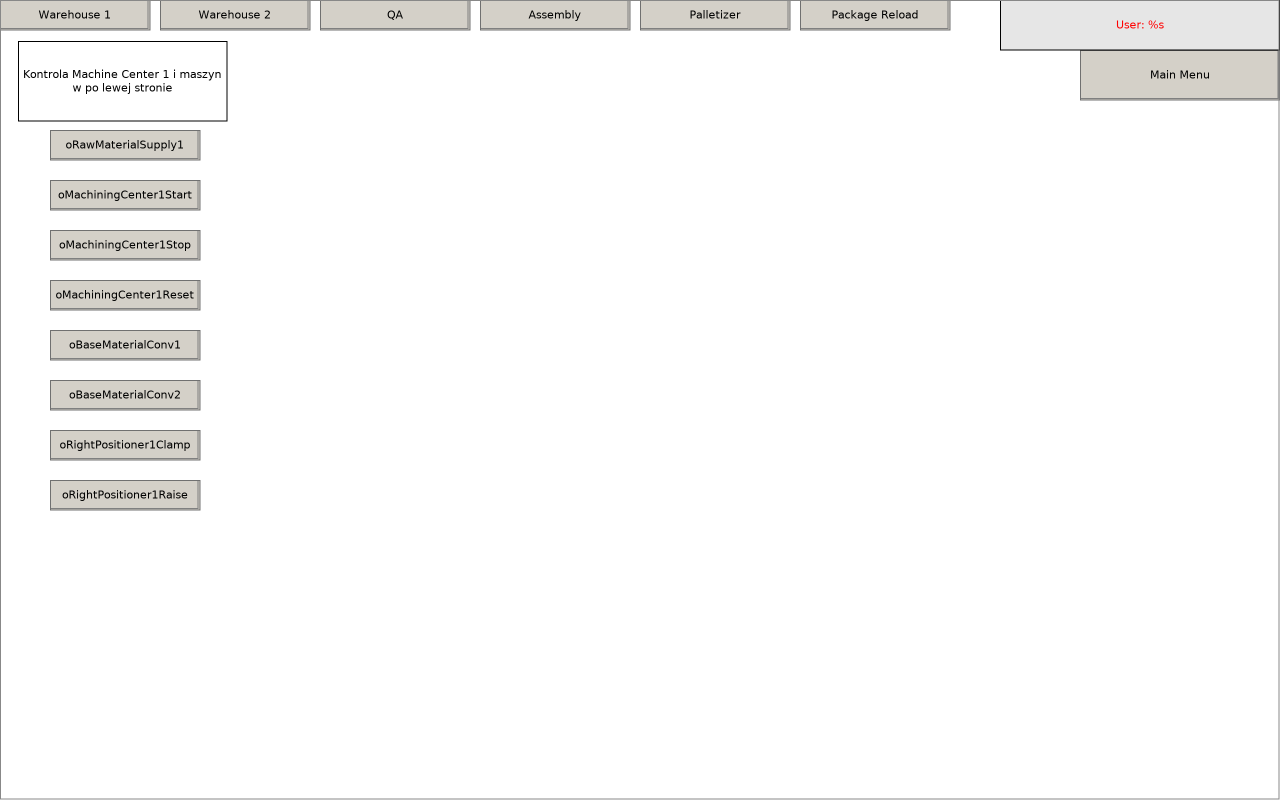
VISUALIZATION Assembly  // 1280x800
    Button (0,0 150x30), "Warehouse 1", colour toggle: HMI.ScreenColor = 1
        OnMouseDown:  Assign=Warehosue_1, Type=Assignment
        OnMouseDown: execute { HMI.ScreenColor := 1; }
    Button (160,0 150x30), "Warehouse 2", colour toggle: HMI.ScreenColor = 2
        OnMouseDown:  Assign=Warehouse_2, Type=Assignment
        OnMouseDown: execute { HMI.ScreenColor := 2; }
    Button (320,0 150x30), "QA", colour toggle: HMI.ScreenColor = 3
        OnMouseDown:  Assign=QA, Type=Assignment
        OnMouseDown: execute { HMI.ScreenColor := 3; }
    Button (480,0 150x30), "Assembly", colour toggle: HMI.ScreenColor = 4
        OnMouseDown:  Assign=Assembly, Type=Assignment
        OnMouseDown: execute { HMI.ScreenColor := 4; }
    Button (640,0 150x30), "Palletizer", colour toggle: HMI.ScreenColor = 5
        OnMouseDown:  Assign=Palletizer, Type=Assignment
        OnMouseDown: execute { HMI.ScreenColor := 5; }
    Button (800,0 150x30), "Package Reload", colour toggle: HMI.ScreenColor = 6
        OnMouseDown:  Assign=Package_Reload, Type=Assignment
        OnMouseDown: execute { HMI.ScreenColor := 6; }
    Button (1080,50 200x50), "Main Menu", colour toggle: HMI.ScreenColor = 0
        OnMouseDown:  Assign=Menu, Type=Assignment
        OnMouseDown: execute { HMI.ScreenColor := 0; }
    Rectangle (1000,0 280x50), "User: %s", text variable: VisuNativeControl.CurrentFullUserName
    Button (50,130 150x30), "oRawMaterialSupply1", invisible if: OPC.iAssemblyAutomatic, input disabled if: OPC.iAssemblyAutomatic
    Rectangle (18,41 209x80), "Kontrola Machine Center 1 i maszyn w po lewej stronie"
    Button (50,180 150x30), "oMachiningCenter1Start", invisible if: OPC.iAssemblyAutomatic, input disabled if: OPC.iAssemblyAutomatic
    Button (50,230 150x30), "oMachiningCenter1Stop", invisible if: OPC.iAssemblyAutomatic, input disabled if: OPC.iAssemblyAutomatic
    Button (50,280 150x30), "oMachiningCenter1Reset", invisible if: OPC.iAssemblyAutomatic, input disabled if: OPC.iAssemblyAutomatic
    Button (50,330 150x30), "oBaseMaterialConv1", invisible if: OPC.iAssemblyAutomatic, input disabled if: OPC.iAssemblyAutomatic
    Button (50,380 150x30), "oBaseMaterialConv2", invisible if: OPC.iAssemblyAutomatic, input disabled if: OPC.iAssemblyAutomatic
    Button (50,430 150x30), "oRightPositioner1Clamp", invisible if: OPC.iAssemblyAutomatic, input disabled if: OPC.iAssemblyAutomatic
    Button (50,480 150x30), "oRightPositioner1Raise", invisible if: OPC.iAssemblyAutomatic, input disabled if: OPC.iAssemblyAutomatic
END_VISUALIZATION

// Device/Application/Menu
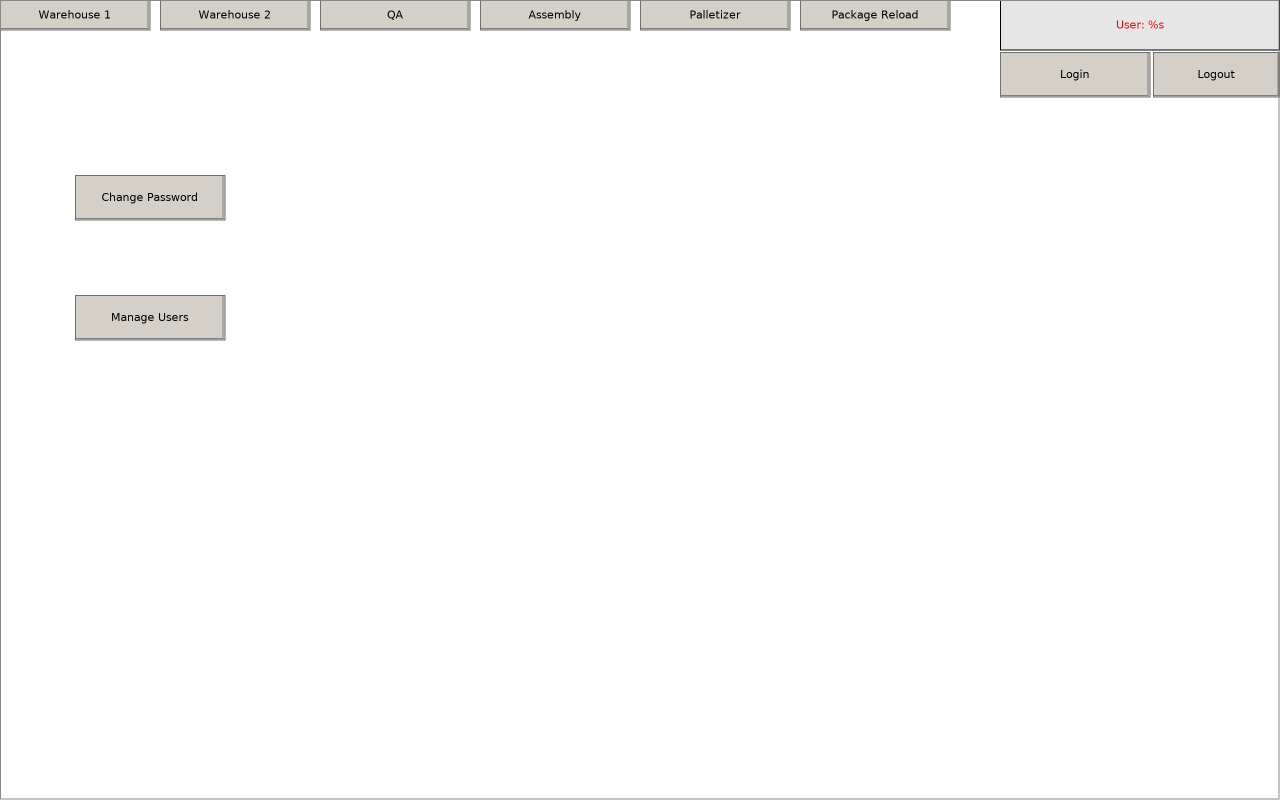
VISUALIZATION Menu  // 1280x800
    Button (0,0 150x30), "Warehouse 1", colour toggle: HMI.ScreenColor = 1
        OnMouseDown:  Assign=Warehosue_1, Type=Assignment
        OnMouseDown: execute { HMI.ScreenColor := 1; }
    Button (160,0 150x30), "Warehouse 2", colour toggle: HMI.ScreenColor = 2
        OnMouseDown:  Assign=Warehouse_2, Type=Assignment
        OnMouseDown: execute { HMI.ScreenColor := 2; }
    Button (320,0 150x30), "QA", colour toggle: HMI.ScreenColor = 3
        OnMouseDown:  Assign=QA, Type=Assignment
        OnMouseDown: execute { HMI.ScreenColor := 3; }
    Button (480,0 150x30), "Assembly", colour toggle: HMI.ScreenColor = 4
        OnMouseDown:  Assign=Assembly, Type=Assignment
        OnMouseDown: execute { HMI.ScreenColor := 4; }
    Button (640,0 150x30), "Palletizer", colour toggle: HMI.ScreenColor = 5
        OnMouseDown:  Assign=Palletizer, Type=Assignment
        OnMouseDown: execute { HMI.ScreenColor := 5; }
    Button (800,0 150x30), "Package Reload", colour toggle: HMI.ScreenColor = 6
        OnMouseDown:  Assign=Package_Reload, Type=Assignment
        OnMouseDown: execute { HMI.ScreenColor := 6; }
    Rectangle (1000,0 280x50), "User: %s", text variable: VisuNativeControl.CurrentFullUserName
    Button (1000,52 150x45), "Login"
        OnMouseDown:  Type=Login
    Button (1153,52 127x45), "Logout"
        OnMouseDown:  Type=Logout
    Button (75,175 150x45), "Change Password"
        OnMouseDown:  Type=ChangeUserPassword
    Button (75,295 150x45), "Manage Users"
        OnMouseDown:  Type=OpenUserConfiguration
END_VISUALIZATION

// Device/Application/Package_Reload
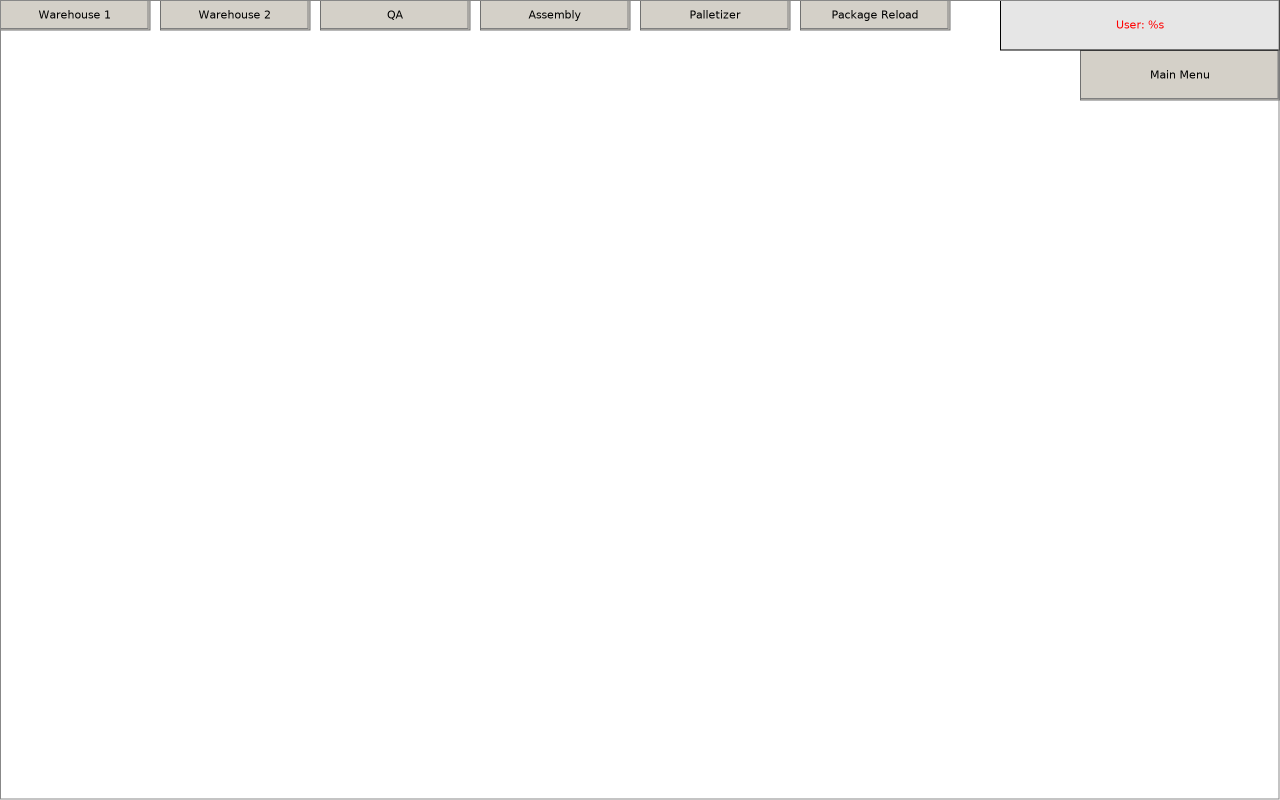
VISUALIZATION Package_Reload  // 1280x800
    Button (0,0 150x30), "Warehouse 1", colour toggle: HMI.ScreenColor = 1
        OnMouseDown:  Assign=Warehosue_1, Type=Assignment
        OnMouseDown: execute { HMI.ScreenColor := 1; }
    Button (160,0 150x30), "Warehouse 2", colour toggle: HMI.ScreenColor = 2
        OnMouseDown:  Assign=Warehouse_2, Type=Assignment
        OnMouseDown: execute { HMI.ScreenColor := 2; }
    Button (320,0 150x30), "QA", colour toggle: HMI.ScreenColor = 3
        OnMouseDown:  Assign=QA, Type=Assignment
        OnMouseDown: execute { HMI.ScreenColor := 3; }
    Button (480,0 150x30), "Assembly", colour toggle: HMI.ScreenColor = 4
        OnMouseDown:  Assign=Assembly, Type=Assignment
        OnMouseDown: execute { HMI.ScreenColor := 4; }
    Button (640,0 150x30), "Palletizer", colour toggle: HMI.ScreenColor = 5
        OnMouseDown:  Assign=Palletizer, Type=Assignment
        OnMouseDown: execute { HMI.ScreenColor := 5; }
    Button (800,0 150x30), "Package Reload", colour toggle: HMI.ScreenColor = 6
        OnMouseDown:  Assign=Package_Reload, Type=Assignment
        OnMouseDown: execute { HMI.ScreenColor := 6; }
    Button (1080,50 200x50), "Main Menu", colour toggle: HMI.ScreenColor = 0
        OnMouseDown:  Assign=Menu, Type=Assignment
        OnMouseDown: execute { HMI.ScreenColor := 0; }
    Rectangle (1000,0 280x50), "User: %s", text variable: VisuNativeControl.CurrentFullUserName
END_VISUALIZATION

// Device/Application/Palletizer
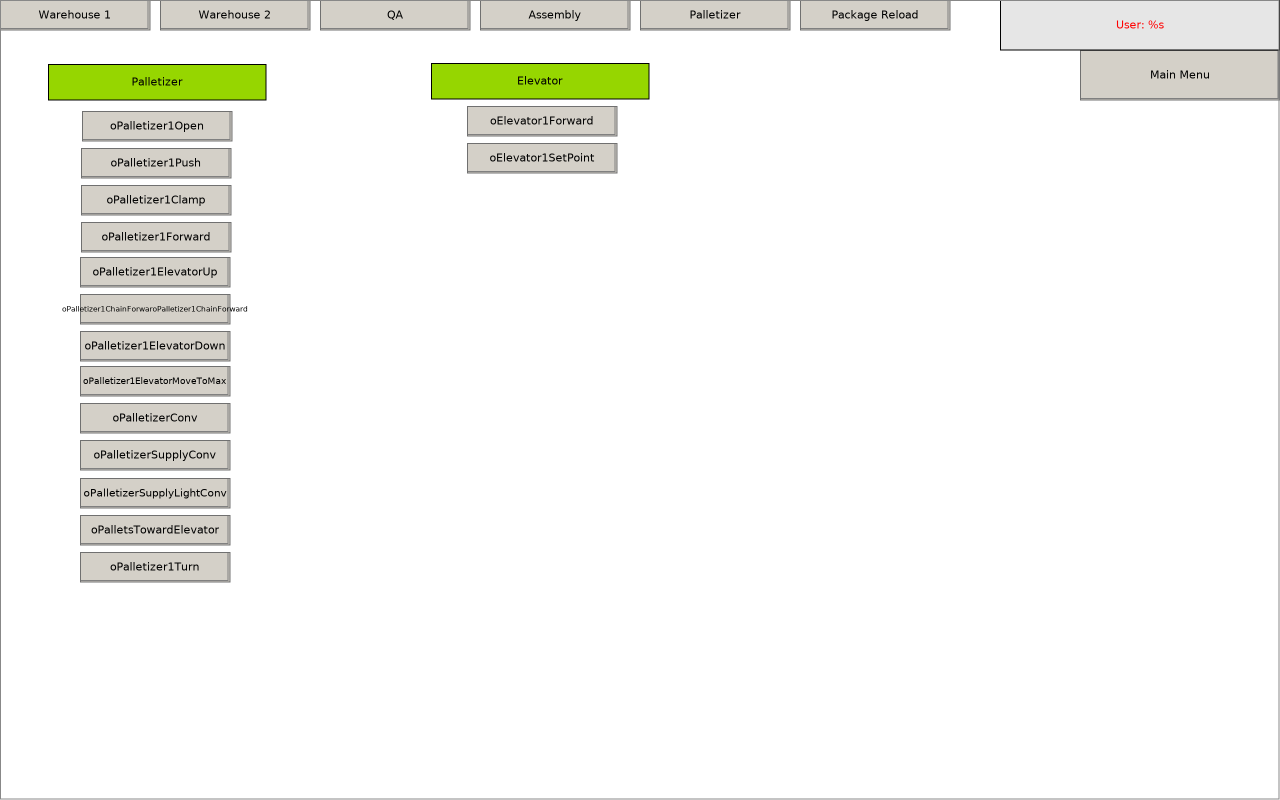
VISUALIZATION Palletizer  // 1280x800
    Button (0,0 150x30), "Warehouse 1", colour toggle: HMI.ScreenColor = 1
        OnMouseDown:  Assign=Warehosue_1, Type=Assignment
        OnMouseDown: execute { HMI.ScreenColor := 1; }
    Button (160,0 150x30), "Warehouse 2", colour toggle: HMI.ScreenColor = 2
        OnMouseDown:  Assign=Warehouse_2, Type=Assignment
        OnMouseDown: execute { HMI.ScreenColor := 2; }
    Button (320,0 150x30), "QA", colour toggle: HMI.ScreenColor = 3
        OnMouseDown:  Assign=QA, Type=Assignment
        OnMouseDown: execute { HMI.ScreenColor := 3; }
    Button (480,0 150x30), "Assembly", colour toggle: HMI.ScreenColor = 4
        OnMouseDown:  Assign=Assembly, Type=Assignment
        OnMouseDown: execute { HMI.ScreenColor := 4; }
    Button (640,0 150x30), "Palletizer", colour toggle: HMI.ScreenColor = 5
        OnMouseDown:  Assign=Palletizer, Type=Assignment
        OnMouseDown: execute { HMI.ScreenColor := 5; }
    Button (800,0 150x30), "Package Reload", colour toggle: HMI.ScreenColor = 6
        OnMouseDown:  Assign=Package_Reload, Type=Assignment
        OnMouseDown: execute { HMI.ScreenColor := 6; }
    Button (1080,50 200x50), "Main Menu", colour toggle: HMI.ScreenColor = 0
        OnMouseDown:  Assign=Menu, Type=Assignment
        OnMouseDown: execute { HMI.ScreenColor := 0; }
    Rectangle (1000,0 280x50), "User: %s", text variable: VisuNativeControl.CurrentFullUserName
    Button (467,106 150x30), "oElevator1Forward", invisible if: OPC.iAssemblyAutomatic, input disabled if: OPC.iAssemblyAutomatic
        toggle HMI.oElevator1Forward
    Button (467,143 150x30), "oElevator1SetPoint", invisible if: OPC.iAssemblyAutomatic, input disabled if: OPC.iAssemblyAutomatic
        toggle OPC.oElevator1SetPoint
    Button (82,111 150x30), "oPalletizer1Open", invisible if: OPC.iAssemblyAutomatic, input disabled if: OPC.iAssemblyAutomatic
        toggle HMI.oPalletizer1Open
    Button (81,148 150x30), "oPalletizer1Push", invisible if: OPC.iAssemblyAutomatic, input disabled if: OPC.iAssemblyAutomatic
        toggle HMI.oPalletizer1Push
    Button (81,185 150x30), "oPalletizer1Clamp", invisible if: OPC.iAssemblyAutomatic, input disabled if: OPC.iAssemblyAutomatic
        toggle HMI.oPalletizer1Clamp
    Button (81,222 150x30), "oPalletizer1Forward", invisible if: OPC.iAssemblyAutomatic, input disabled if: OPC.iAssemblyAutomatic
        toggle HMI.oPalletizer1Forward
    Button (80,257 150x30), "oPalletizer1ElevatorUp", invisible if: OPC.iAssemblyAutomatic, input disabled if: OPC.iAssemblyAutomatic
        toggle HMI.oPalletizer1ElevatorUp
    Button (80,294 150x30), "oPalletizer1ChainForwaroPalletizer1ChainForward", invisible if: OPC.iAssemblyAutomatic, input disabled if: OPC.iAssemblyAutomatic
        toggle HMI.oPalletizer1ChainForward
    Button (80,331 150x30), "oPalletizer1ElevatorDown", invisible if: OPC.iAssemblyAutomatic, input disabled if: OPC.iAssemblyAutomatic
        toggle HMI.oPalletizer1ElevatorDown
    Button (80,366 150x30), "oPalletizer1ElevatorMoveToMax", invisible if: OPC.iAssemblyAutomatic, input disabled if: OPC.iAssemblyAutomatic
        toggle HMI.oPalletizer1ElevatorMoveToMax
    Button (80,403 150x30), "oPalletizerConv", invisible if: OPC.iAssemblyAutomatic, input disabled if: OPC.iAssemblyAutomatic
        toggle HMI.oPalletizerConv
    Button (80,440 150x30), "oPalletizerSupplyConv", invisible if: OPC.iAssemblyAutomatic, input disabled if: OPC.iAssemblyAutomatic
        toggle HMI.oPalletizerSupplyConv
    Button (80,478 150x30), "oPalletizerSupplyLightConv", invisible if: OPC.iAssemblyAutomatic, input disabled if: OPC.iAssemblyAutomatic
        toggle HMI.oPalletizerSupplyLightConv
    Button (80,515 150x30), "oPalletsTowardElevator", invisible if: OPC.iAssemblyAutomatic, input disabled if: OPC.iAssemblyAutomatic
        toggle HMI.oPalletsTowardElevator
    Button (80,552 150x30), "oPalletizer1Turn", invisible if: OPC.iAssemblyAutomatic, input disabled if: OPC.iAssemblyAutomatic
        toggle HMI.oPalletizer1Turn
    Rectangle (431,63 218x36), "Elevator"
    Rectangle (48,64 218x36), "Palletizer"
END_VISUALIZATION

// Device/Application/QA
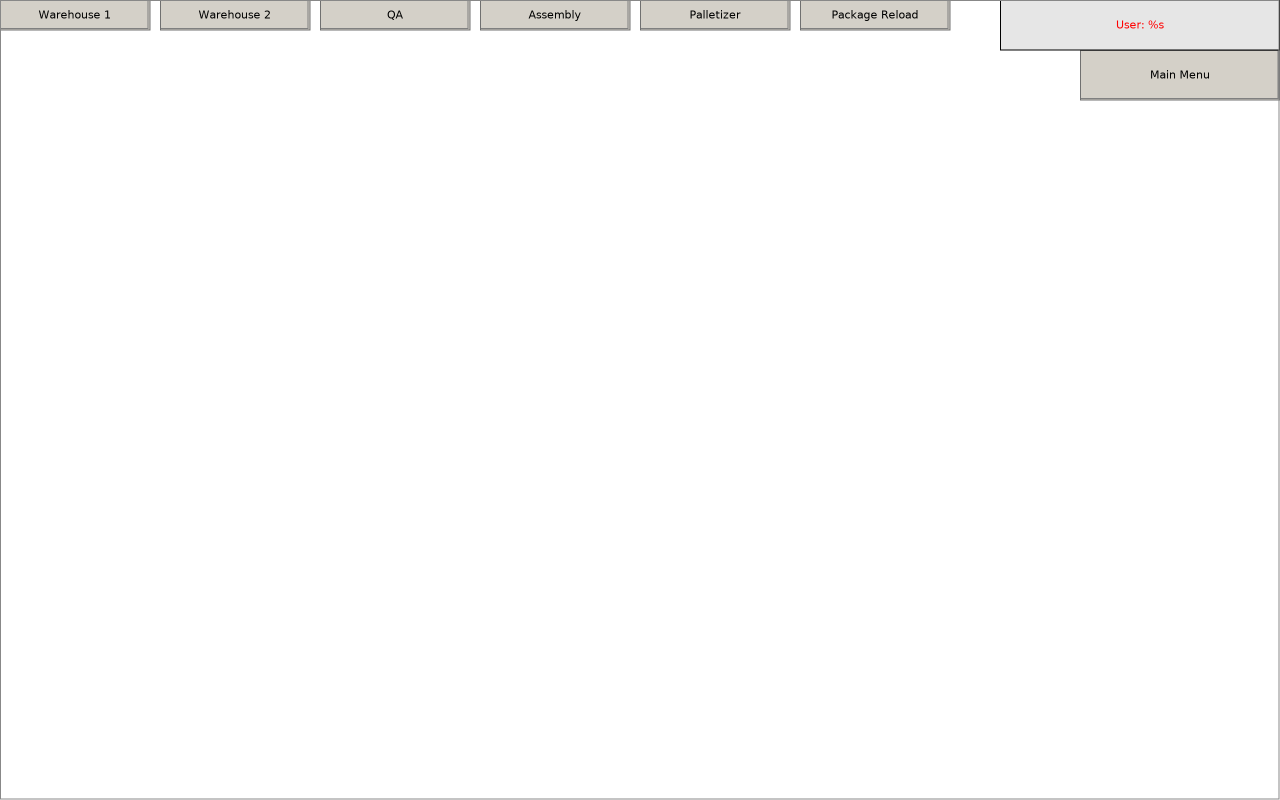
VISUALIZATION QA  // 1280x800
    Button (0,0 150x30), "Warehouse 1", colour toggle: HMI.ScreenColor = 1
        OnMouseDown:  Assign=Warehosue_1, Type=Assignment
        OnMouseDown: execute { HMI.ScreenColor := 1; }
    Button (160,0 150x30), "Warehouse 2", colour toggle: HMI.ScreenColor = 2
        OnMouseDown:  Assign=Warehouse_2, Type=Assignment
        OnMouseDown: execute { HMI.ScreenColor := 2; }
    Button (320,0 150x30), "QA", colour toggle: HMI.ScreenColor = 3
        OnMouseDown:  Assign=QA, Type=Assignment
        OnMouseDown: execute { HMI.ScreenColor := 3; }
    Button (480,0 150x30), "Assembly", colour toggle: HMI.ScreenColor = 4
        OnMouseDown:  Assign=Assembly, Type=Assignment
        OnMouseDown: execute { HMI.ScreenColor := 4; }
    Button (640,0 150x30), "Palletizer", colour toggle: HMI.ScreenColor = 5
        OnMouseDown:  Assign=Palletizer, Type=Assignment
        OnMouseDown: execute { HMI.ScreenColor := 5; }
    Button (800,0 150x30), "Package Reload", colour toggle: HMI.ScreenColor = 6
        OnMouseDown:  Assign=Package_Reload, Type=Assignment
        OnMouseDown: execute { HMI.ScreenColor := 6; }
    Button (1080,50 200x50), "Main Menu", colour toggle: HMI.ScreenColor = 0
        OnMouseDown:  Assign=Menu, Type=Assignment
        OnMouseDown: execute { HMI.ScreenColor := 0; }
    Rectangle (1000,0 280x50), "User: %s", text variable: VisuNativeControl.CurrentFullUserName
END_VISUALIZATION

// Device/Application/Warehosue_1
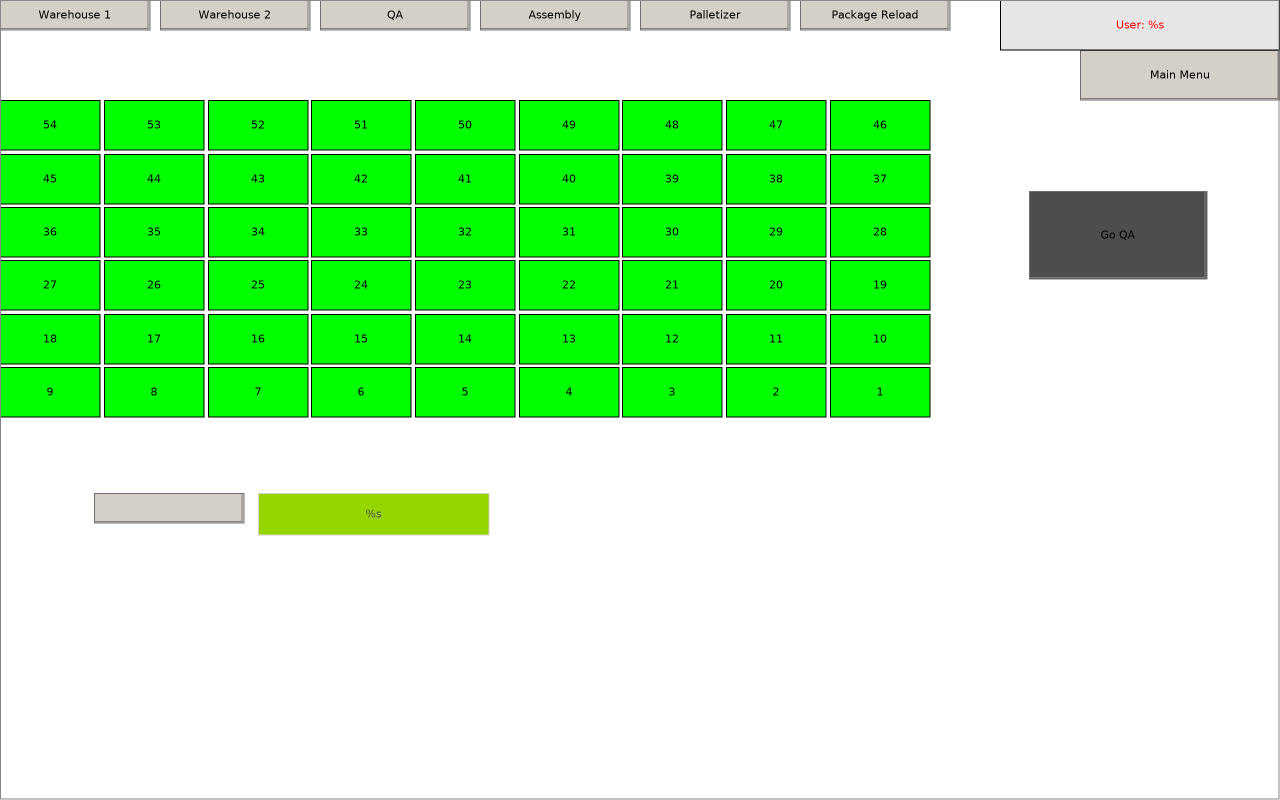
VISUALIZATION Warehosue_1  // 1280x800
    Rectangle (0,100 100x50), "54", colour toggle: GVL.Warehouse1Array[54] = 1
    Rectangle (104,100 100x50), "53", colour toggle: GVL.Warehouse1Array[53] = 1
    Rectangle (208,100 100x50), "52", colour toggle: GVL.Warehouse1Array[52] = 1
    Rectangle (311,100 100x50), "51", colour toggle: GVL.Warehouse1Array[51] = 1
    Rectangle (415,100 100x50), "50", colour toggle: GVL.Warehouse1Array[50] = 1
    Rectangle (519,100 100x50), "49", colour toggle: GVL.Warehouse1Array[49] = 1
    Rectangle (622,100 100x50), "48", colour toggle: GVL.Warehouse1Array[48] = 1
    Rectangle (726,100 100x50), "47", colour toggle: GVL.Warehouse1Array[47] = 1
    Rectangle (830,100 100x50), "46", colour toggle: GVL.Warehouse1Array[46] = 1
    Rectangle (0,154 100x50), "45", colour toggle: GVL.Warehouse1Array[45] = 1
    Rectangle (104,154 100x50), "44", colour toggle: GVL.Warehouse1Array[44] = 1
    Rectangle (208,154 100x50), "43", colour toggle: GVL.Warehouse1Array[43] = 1
    Rectangle (311,154 100x50), "42", colour toggle: GVL.Warehouse1Array[42] = 1
    Rectangle (415,154 100x50), "41", colour toggle: GVL.Warehouse1Array[41] = 1
    Rectangle (519,154 100x50), "40", colour toggle: GVL.Warehouse1Array[40] = 1
    Rectangle (622,154 100x50), "39", colour toggle: GVL.Warehouse1Array[39] = 1
    Rectangle (726,154 100x50), "38", colour toggle: GVL.Warehouse1Array[35] = 1
    Rectangle (830,154 100x50), "37", colour toggle: GVL.Warehouse1Array[37] = 1
    Rectangle (0,207 100x50), "36", colour toggle: GVL.Warehouse1Array[36] = 1
    Rectangle (104,207 100x50), "35", colour toggle: GVL.Warehouse1Array[35] = 1
    Rectangle (208,207 100x50), "34", colour toggle: GVL.Warehouse1Array[34] = 1
    Rectangle (311,207 100x50), "33", colour toggle: GVL.Warehouse1Array[33] = 1
    Rectangle (415,207 100x50), "32", colour toggle: GVL.Warehouse1Array[32] = 1
    Rectangle (519,207 100x50), "31", colour toggle: GVL.Warehouse1Array[31] = 1
    Rectangle (622,207 100x50), "30", colour toggle: GVL.Warehouse1Array[23] = 1
    Rectangle (726,207 100x50), "29", colour toggle: GVL.Warehouse1Array[29] = 1
    Rectangle (830,207 100x50), "28", colour toggle: GVL.Warehouse1Array[28] = 1
    Rectangle (0,260 100x50), "27", colour toggle: GVL.Warehouse1Array[27] = 1
    Rectangle (104,260 100x50), "26", colour toggle: GVL.Warehouse1Array[26] = 1
    Rectangle (208,260 100x50), "25", colour toggle: GVL.Warehouse1Array[25] = 1
    Rectangle (311,260 100x50), "24", colour toggle: GVL.Warehouse1Array[24] = 1
    Rectangle (415,260 100x50), "23", colour toggle: GVL.Warehouse1Array[23] = 1
    Rectangle (519,260 100x50), "22", colour toggle: GVL.Warehouse1Array[22] = 1
    Rectangle (622,260 100x50), "21", colour toggle: GVL.Warehouse1Array[21] = 1
    Rectangle (726,260 100x50), "20", colour toggle: GVL.Warehouse1Array[20] = 1
    Rectangle (830,260 100x50), "19", colour toggle: GVL.Warehouse1Array[19] = 1
    Rectangle (0,314 100x50), "18", colour toggle: GVL.Warehouse1Array[18] = 1
    Rectangle (104,314 100x50), "17", colour toggle: GVL.Warehouse1Array[17] = 1
    Rectangle (208,314 100x50), "16", colour toggle: GVL.Warehouse1Array[16] = 1
    Rectangle (311,314 100x50), "15", colour toggle: GVL.Warehouse1Array[15] = 1
    Rectangle (415,314 100x50), "14", colour toggle: GVL.Warehouse1Array[14] = 1
    Rectangle (519,314 100x50), "13", colour toggle: GVL.Warehouse1Array[13] = 1
    Rectangle (622,314 100x50), "12", colour toggle: GVL.Warehouse1Array[12] = 1
    Rectangle (726,314 100x50), "11", colour toggle: GVL.Warehouse1Array[11] = 1
    Rectangle (830,314 100x50), "10", colour toggle: GVL.Warehouse1Array[10] = 1
    Rectangle (0,367 100x50), "9", colour toggle: GVL.Warehouse1Array[9] = 1
    Rectangle (104,367 100x50), "8", colour toggle: GVL.Warehouse1Array[8] = 1
    Rectangle (208,367 100x50), "7", colour toggle: GVL.Warehouse1Array[7] = 1
    Rectangle (311,367 100x50), "6", colour toggle: GVL.Warehouse1Array[6] = 1
    Rectangle (415,367 100x50), "5", colour toggle: GVL.Warehouse1Array[5] = 1
    Rectangle (519,367 100x50), "4", colour toggle: GVL.Warehouse1Array[4] = 1
    Rectangle (622,367 100x50), "3", colour toggle: GVL.Warehouse1Array[3] = 1
    Rectangle (726,367 100x50), "2", colour toggle: GVL.Warehouse1Array[2] = 1
    Rectangle (830,367 100x50), "1", colour toggle: GVL.Warehouse1Array[1] = 1
    Button (1029,191 178x88), "Go QA", colour toggle: HMI.GoingQA
        toggle HMI.GoingQA
    Button (0,0 150x30), "Warehouse 1", colour toggle: HMI.ScreenColor = 1
        OnMouseDown:  Assign=Warehosue_1, Type=Assignment
        OnMouseDown: execute { HMI.ScreenColor := 1; }
    Button (160,0 150x30), "Warehouse 2", colour toggle: HMI.ScreenColor = 2
        OnMouseDown:  Assign=Warehouse_2, Type=Assignment
        OnMouseDown: execute { HMI.ScreenColor := 2; }
    Button (320,0 150x30), "QA", colour toggle: HMI.ScreenColor = 3
        OnMouseDown:  Assign=QA, Type=Assignment
        OnMouseDown: execute { HMI.ScreenColor := 3; }
    Button (480,0 150x30), "Assembly", colour toggle: HMI.ScreenColor = 4
        OnMouseDown:  Assign=Assembly, Type=Assignment
        OnMouseDown: execute { HMI.ScreenColor := 4; }
    Button (640,0 150x30), "Palletizer", colour toggle: HMI.ScreenColor = 5
        OnMouseDown:  Assign=Palletizer, Type=Assignment
        OnMouseDown: execute { HMI.ScreenColor := 5; }
    Button (800,0 150x30), "Package Reload", colour toggle: HMI.ScreenColor = 6
        OnMouseDown:  Assign=Package_Reload, Type=Assignment
        OnMouseDown: execute { HMI.ScreenColor := 6; }
    Button (1080,50 200x50), "Main Menu", colour toggle: HMI.ScreenColor = 0
        OnMouseDown:  Assign=Menu, Type=Assignment
        OnMouseDown: execute { HMI.ScreenColor := 0; }
    Rectangle (1000,0 280x50), "User: %s", text variable: VisuNativeControl.CurrentFullUserName
    Button (94,493 150x30)
        toggle HMI.Pick1
    Textfield (258,493 231x42), "%s", text variable: HMI.WantedMaterial1
END_VISUALIZATION

// Device/Application/Warehouse_2
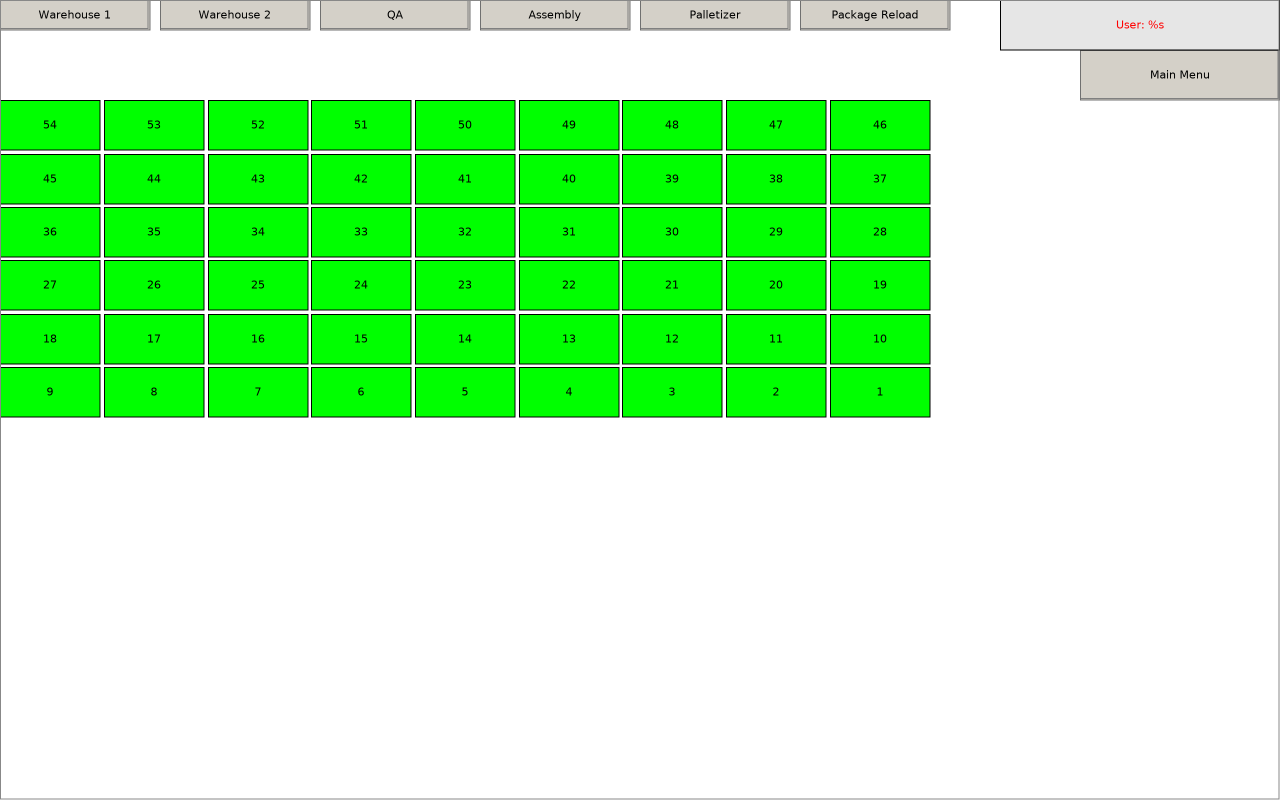
VISUALIZATION Warehouse_2  // 1280x800
    Button (0,0 150x30), "Warehouse 1", colour toggle: HMI.ScreenColor = 1
        OnMouseDown:  Assign=Warehosue_1, Type=Assignment
        OnMouseDown: execute { HMI.ScreenColor := 1; }
    Button (160,0 150x30), "Warehouse 2", colour toggle: HMI.ScreenColor = 2
        OnMouseDown:  Assign=Warehouse_2, Type=Assignment
        OnMouseDown: execute { HMI.ScreenColor := 2; }
    Button (320,0 150x30), "QA", colour toggle: HMI.ScreenColor = 3
        OnMouseDown:  Assign=QA, Type=Assignment
        OnMouseDown: execute { HMI.ScreenColor := 3; }
    Button (480,0 150x30), "Assembly", colour toggle: HMI.ScreenColor = 4
        OnMouseDown:  Assign=Assembly, Type=Assignment
        OnMouseDown: execute { HMI.ScreenColor := 4; }
    Button (640,0 150x30), "Palletizer", colour toggle: HMI.ScreenColor = 5
        OnMouseDown:  Assign=Palletizer, Type=Assignment
        OnMouseDown: execute { HMI.ScreenColor := 5; }
    Button (800,0 150x30), "Package Reload", colour toggle: HMI.ScreenColor = 6
        OnMouseDown:  Assign=Package_Reload, Type=Assignment
        OnMouseDown: execute { HMI.ScreenColor := 6; }
    Button (1080,50 200x50), "Main Menu", colour toggle: HMI.ScreenColor = 0
        OnMouseDown:  Assign=Menu, Type=Assignment
        OnMouseDown: execute { HMI.ScreenColor := 0; }
    Rectangle (1000,0 280x50), "User: %s", text variable: VisuNativeControl.CurrentFullUserName
    Rectangle (0,100 100x50), "54", colour toggle: GVL.Warehouse2Array[54] = 1
    Rectangle (104,100 100x50), "53", colour toggle: GVL.Warehouse2Array[53] = 1
    Rectangle (208,100 100x50), "52", colour toggle: GVL.Warehouse2Array[52] = 1
    Rectangle (311,100 100x50), "51", colour toggle: GVL.Warehouse2Array[51] = 1
    Rectangle (415,100 100x50), "50", colour toggle: GVL.Warehouse2Array[50] = 1
    Rectangle (519,100 100x50), "49", colour toggle: GVL.Warehouse2Array[49] = 1
    Rectangle (622,100 100x50), "48", colour toggle: GVL.Warehouse2Array[48] = 1
    Rectangle (726,100 100x50), "47", colour toggle: GVL.Warehouse2Array[47] = 1
    Rectangle (830,100 100x50), "46", colour toggle: GVL.Warehouse2Array[46] = 1
    Rectangle (0,154 100x50), "45", colour toggle: GVL.Warehouse2Array[45] = 1
    Rectangle (104,154 100x50), "44", colour toggle: GVL.Warehouse2Array[44] = 1
    Rectangle (208,154 100x50), "43", colour toggle: GVL.Warehouse2Array[43] = 1
    Rectangle (311,154 100x50), "42", colour toggle: GVL.Warehouse2Array[42] = 1
    Rectangle (415,154 100x50), "41", colour toggle: GVL.Warehouse2Array[41] = 1
    Rectangle (519,154 100x50), "40", colour toggle: GVL.Warehouse2Array[40] = 1
    Rectangle (622,154 100x50), "39", colour toggle: GVL.Warehouse2Array[39] = 1
    Rectangle (726,154 100x50), "38", colour toggle: GVL.Warehouse2Array[35] = 1
    Rectangle (830,154 100x50), "37", colour toggle: GVL.Warehouse2Array[37] = 1
    Rectangle (0,207 100x50), "36", colour toggle: GVL.Warehouse2Array[36] = 1
    Rectangle (104,207 100x50), "35", colour toggle: GVL.Warehouse2Array[35] = 1
    Rectangle (208,207 100x50), "34", colour toggle: GVL.Warehouse2Array[34] = 1
    Rectangle (311,207 100x50), "33", colour toggle: GVL.Warehouse2Array[33] = 1
    Rectangle (415,207 100x50), "32", colour toggle: GVL.Warehouse2Array[32] = 1
    Rectangle (519,207 100x50), "31", colour toggle: GVL.Warehouse2Array[31] = 1
    Rectangle (622,207 100x50), "30", colour toggle: GVL.Warehouse2Array[23] = 1
    Rectangle (726,207 100x50), "29", colour toggle: GVL.Warehouse2Array[29] = 1
    Rectangle (830,207 100x50), "28", colour toggle: GVL.Warehouse2Array[28] = 1
    Rectangle (0,260 100x50), "27", colour toggle: GVL.Warehouse2Array[27] = 1
    Rectangle (104,260 100x50), "26", colour toggle: GVL.Warehouse2Array[26] = 1
    Rectangle (208,260 100x50), "25", colour toggle: GVL.Warehouse2Array[25] = 1
    Rectangle (311,260 100x50), "24", colour toggle: GVL.Warehouse2Array[24] = 1
    Rectangle (415,260 100x50), "23", colour toggle: GVL.Warehouse2Array[23] = 1
    Rectangle (519,260 100x50), "22", colour toggle: GVL.Warehouse2Array[22] = 1
    Rectangle (622,260 100x50), "21", colour toggle: GVL.Warehouse2Array[21] = 1
    Rectangle (726,260 100x50), "20", colour toggle: GVL.Warehouse2Array[20] = 1
    Rectangle (830,260 100x50), "19", colour toggle: GVL.Warehouse2Array[19] = 1
    Rectangle (0,314 100x50), "18", colour toggle: GVL.Warehouse2Array[18] = 1
    Rectangle (104,314 100x50), "17", colour toggle: GVL.Warehouse2Array[17] = 1
    Rectangle (208,314 100x50), "16", colour toggle: GVL.Warehouse2Array[16] = 1
    Rectangle (311,314 100x50), "15", colour toggle: GVL.Warehouse2Array[15] = 1
    Rectangle (415,314 100x50), "14", colour toggle: GVL.Warehouse2Array[14] = 1
    Rectangle (519,314 100x50), "13", colour toggle: GVL.Warehouse2Array[13] = 1
    Rectangle (622,314 100x50), "12", colour toggle: GVL.Warehouse2Array[12] = 1
    Rectangle (726,314 100x50), "11", colour toggle: GVL.Warehouse2Array[11] = 1
    Rectangle (830,314 100x50), "10", colour toggle: GVL.Warehouse2Array[10] = 1
    Rectangle (0,367 100x50), "9", colour toggle: GVL.Warehouse2Array[9] = 1
    Rectangle (104,367 100x50), "8", colour toggle: GVL.Warehouse2Array[8] = 1
    Rectangle (208,367 100x50), "7", colour toggle: GVL.Warehouse2Array[7] = 1
    Rectangle (311,367 100x50), "6", colour toggle: GVL.Warehouse2Array[6] = 1
    Rectangle (415,367 100x50), "5", colour toggle: GVL.Warehouse2Array[5] = 1
    Rectangle (519,367 100x50), "4", colour toggle: GVL.Warehouse2Array[4] = 1
    Rectangle (622,367 100x50), "3", colour toggle: GVL.Warehouse2Array[3] = 1
    Rectangle (726,367 100x50), "2", colour toggle: GVL.Warehouse2Array[2] = 1
    Rectangle (830,367 100x50), "1", colour toggle: GVL.Warehouse2Array[1] = 1
END_VISUALIZATION
